KUKA KRL program: MyProgram_133().src

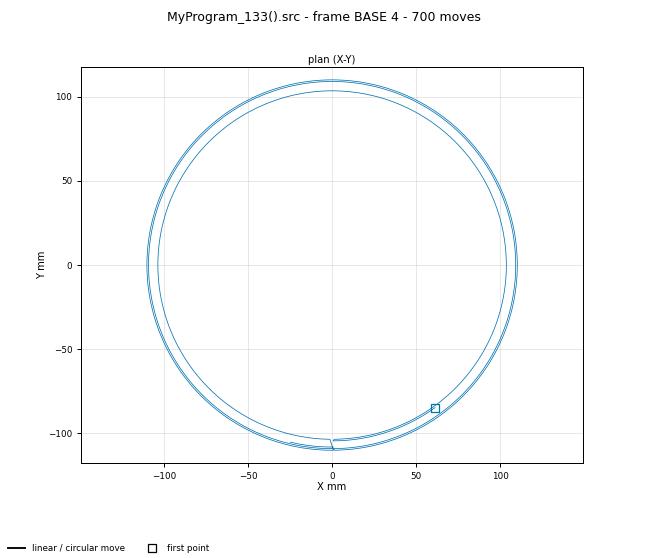
[picture p0: tool path of MyProgram_133().src in frame BASE 4, 700 of 700 moves have a stored position in this frame; points joined in program order, loops and branches not executed]
&ACCESS RVP
&REL 1
&PARAM TEMPLATE = C:\KRC\Roboter\Template\vorgabe
&PARAM EDITMASK = *
DEF MyProgram_133()
; ---- Setting reference (Base) ----
$BASE = BASE_DATA[4]

; --------------------------
; ---- Setting tool (TCP) ----
$TOOL = TOOL_DATA[3]
; --------------------------

$VEL.CP = VEL_APROX_PRINT
Startdeposition()
$VEL.CP = VEL_PRINT
LIN {X 61.2206,Y -84.8181,Z 108,A -58.6643,B 24.9452,C -1.7099,E1 25.0928,E2 504.3174} C_DIS
LIN {X 58.1513,Y -86.9519,Z 108,A -60.6312,B 24.9452,C -1.7091,E1 25.0883,E2 506.2796} C_DIS
LIN {X 55.4744,Y -88.6817,Z 108,A -62.4404,B 24.9456,C -1.7031,E1 25.084,E2 508.097} C_DIS
LIN {X 52.3012,Y -90.5896,Z 108,A -64.1698,B 24.9451,C -1.7116,E1 25.0799,E2 509.801} C_DIS
LIN {X 49.6243,Y -92.0835,Z 108,A -66.2153,B 24.9462,C -1.6936,E1 25.0748,E2 511.883} C_DIS
LIN {X 46.4014,Y -93.7484,Z 108,A -67.8646,B 24.9456,C -1.7041,E1 25.0708,E2 513.5031} C_DIS
LIN {X 42.0494,Y -95.7798,Z 108,A -71.2268,B 24.9477,C -1.6704,E1 25.0621,E2 516.9366} C_DIS
LIN {X 38.7203,Y -97.1743,Z 108,A -72.8071,B 24.9469,C -1.6835,E1 25.0581,E2 518.4823} C_DIS
LIN {X 33.6677,Y -99.0374,Z 108,A -75.7053,B 24.947,C -1.6817,E1 25.0505,E2 521.3787} C_DIS
LIN {X 30.0797,Y -100.1857,Z 108,A -77.6032,B 24.9467,C -1.6859,E1 25.0454,E2 523.2633} C_DIS
LIN {X 26.6603,Y -101.1508,Z 108,A -80.0703,B 24.9482,C -1.663,E1 25.0386,E2 525.7807} C_DIS
LIN {X 21.8993,Y -102.286,Z 108,A -82.3229,B 24.9473,C -1.6775,E1 25.0326,E2 527.9957} C_DIS
LIN {X 18.813,Y -102.8981,Z 108,A -84.0847,B 24.9475,C -1.6746,E1 25.0278,E2 529.7625} C_DIS
LIN {X 14.7921,Y -103.5522,Z 108,A -86.2883,B 24.9475,C -1.6741,E1 25.0217,E2 531.9652} C_DIS
LIN {X 12.4769,Y -103.857,Z 108,A -87.7945,B 24.9481,C -1.6643,E1 25.0174,E2 533.4935} C_DIS
LIN {X 8.4641,Y -104.2604,Z 108,A -89.7441,B 24.9475,C -1.6734,E1 25.0121,E2 535.4204} C_DIS
LIN {X 5.3432,Y -104.4676,Z 108,A -91.7149,B 24.9482,C -1.6625,E1 25.0065,E2 537.4162} C_DIS
LIN {X 0.6861,Y -104.5966,Z 108,A -93.2357,B 24.9457,C -1.7025,E1 25.0026,E2 538.842} C_DIS
Enddeposition()
LIN {X 0.6861,Y -104.5966,Z 108,A -93.2357,B 24.9457,C -1.7025,E1 25.0026,E2 538.842} C_DIS
Startdeposition()
$VEL.CP = VEL_PRINT
LIN {X 1.232,Y -103.6397,Z 108,A -93.0353,B 24.9449,C -1.715,E1 25.0032,E2 538.6119} C_DIS
LIN {X 3.4523,Y -103.5881,Z 108,A -91.8043,B 24.9449,C -1.7156,E1 25.0066,E2 537.3798} C_DIS
LIN {X 6.3528,Y -103.4523,Z 108,A -90.1987,B 24.9449,C -1.7162,E1 25.0111,E2 535.7733} C_DIS
LIN {X 8.6388,Y -103.2853,Z 108,A -88.9124,B 24.9447,C -1.7176,E1 25.0147,E2 534.4842} C_DIS
LIN {X 11.1011,Y -103.0495,Z 108,A -87.536,B 24.9447,C -1.7188,E1 25.0185,E2 533.1061} C_DIS
LIN {X 13.6424,Y -102.744,Z 108,A -86.1543,B 24.9447,C -1.7183,E1 25.0223,E2 531.7265} C_DIS
LIN {X 16.4463,Y -102.334,Z 108,A -84.5923,B 24.9447,C -1.7193,E1 25.0267,E2 530.1638} C_DIS
LIN {X 18.9681,Y -101.8968,Z 108,A -83.1777,B 24.9445,C -1.7204,E1 25.0305,E2 528.7481} C_DIS
LIN {X 21.1597,Y -101.4629,Z 108,A -81.9382,B 24.9445,C -1.7217,E1 25.0339,E2 527.5071} C_DIS
LIN {X 23.6339,Y -100.9152,Z 108,A -80.5472,B 24.9444,C -1.7226,E1 25.0377,E2 526.1158} C_DIS
LIN {X 26.3836,Y -100.2328,Z 108,A -78.9876,B 24.9444,C -1.7239,E1 25.0419,E2 524.5554} C_DIS
LIN {X 28.8655,Y -99.5466,Z 108,A -77.564,B 24.9442,C -1.7255,E1 25.0458,E2 523.1304} C_DIS
LIN {X 31.0076,Y -98.8988,Z 108,A -76.33,B 24.9442,C -1.7269,E1 25.0491,E2 521.8955} C_DIS
LIN {X 33.7061,Y -98.0134,Z 108,A -74.7661,B 24.944,C -1.7286,E1 25.0532,E2 520.3305} C_DIS
LIN {X 36.1212,Y -97.1493,Z 108,A -73.3546,B 24.9439,C -1.7302,E1 25.0569,E2 518.9182} C_DIS
LIN {X 38.4749,Y -96.2415,Z 108,A -71.9598,B 24.9438,C -1.7321,E1 25.0605,E2 517.5219} C_DIS
LIN {X 40.5286,Y -95.3932,Z 108,A -70.7044,B 24.9436,C -1.7351,E1 25.0638,E2 516.2624} C_DIS
LIN {X 42.8319,Y -94.3814,Z 108,A -69.3162,B 24.9434,C -1.7371,E1 25.0673,E2 514.8729} C_DIS
LIN {X 45.3665,Y -93.1907,Z 108,A -67.8221,B 24.9434,C -1.7374,E1 25.0711,E2 513.382} C_DIS
LIN {X 47.7293,Y -92.0036,Z 108,A -66.2293,B 24.9429,C -1.7452,E1 25.0751,E2 511.7751} C_DIS
LIN {X 50.5152,Y -90.5017,Z 108,A -64.5337,B 24.9429,C -1.7461,E1 25.0792,E2 510.0823} C_DIS
LIN {X 53.2884,Y -88.8993,Z 108,A -62.8451,B 24.9429,C -1.7459,E1 25.0833,E2 508.3992} C_DIS
LIN {X 55.1927,Y -87.7281,Z 108,A -61.613,B 24.9427,C -1.7482,E1 25.0862,E2 507.1658} C_DIS
LIN {X 57.3228,Y -86.3513,Z 108,A -60.1865,B 24.9425,C -1.7519,E1 25.0895,E2 505.7351} C_DIS
LIN {X 59.6652,Y -84.7513,Z 108,A -58.655,B 24.9424,C -1.7536,E1 25.0931,E2 504.205} C_DIS
LIN {X 61.4771,Y -83.4446,Z 108,A -57.3239,B 24.9419,C -1.7602,E1 25.0961,E2 502.863} C_DIS
LIN {X 64.262,Y -81.3187,Z 108,A -55.4103,B 24.9417,C -1.7634,E1 25.1003,E2 500.9488} C_DIS
LIN {X 67.0825,Y -79.0083,Z 108,A -53.4504,B 24.9416,C -1.7656,E1 25.1045,E2 498.9912} C_DIS
LIN {X 69.5666,Y -76.8321,Z 108,A -51.4729,B 24.9409,C -1.7762,E1 25.1087,E2 496.9967} C_DIS
LIN {X 71.9263,Y -74.6254,Z 108,A -49.8665,B 24.9411,C -1.773,E1 25.1119,E2 495.4045} C_DIS
LIN {X 74.2699,Y -72.2952,Z 108,A -47.9241,B 24.9405,C -1.7823,E1 25.1157,E2 493.4484} C_DIS
LIN {X 76.6554,Y -69.7601,Z 108,A -45.996,B 24.9401,C -1.7873,E1 25.1194,E2 491.5168} C_DIS
LIN {X 78.8973,Y -67.2128,Z 108,A -44.2153,B 24.9401,C -1.7882,E1 25.1226,E2 489.7421} C_DIS
LIN {X 81.2145,Y -64.394,Z 108,A -42.2551,B 24.9399,C -1.7912,E1 25.1261,E2 487.7839} C_DIS
LIN {X 83.0501,Y -62.009,Z 108,A -40.6111,B 24.9396,C -1.7949,E1 25.1288,E2 486.1391} C_DIS
LIN {X 85.1534,Y -59.0868,Z 108,A -38.619,B 24.9392,C -1.8005,E1 25.1321,E2 484.1435} C_DIS
LIN {X 86.8773,Y -56.525,Z 108,A -36.9669,B 24.9391,C -1.8029,E1 25.1346,E2 482.4938} C_DIS
LIN {X 88.5467,Y -53.8686,Z 108,A -35.1672,B 24.9385,C -1.8107,E1 25.1373,E2 480.6849} C_DIS
LIN {X 90.0257,Y -51.3597,Z 108,A -33.6723,B 24.9385,C -1.8105,E1 25.1393,E2 479.1981} C_DIS
LIN {X 91.265,Y -49.1238,Z 108,A -32.2106,B 24.9381,C -1.8168,E1 25.1413,E2 477.7294} C_DIS
LIN {X 92.441,Y -46.8734,Z 108,A -30.8154,B 24.9379,C -1.8206,E1 25.1431,E2 476.3325} C_DIS
LIN {X 93.5614,Y -44.595,Z 108,A -29.2927,B 24.9372,C -1.8298,E1 25.1449,E2 474.7962} C_DIS
LIN {X 95.0266,Y -41.3799,Z 108,A -27.4161,B 24.9371,C -1.8326,E1 25.1471,E2 472.9234} C_DIS
LIN {X 96.1166,Y -38.7819,Z 108,A -25.9637,B 24.9371,C -1.8329,E1 25.1486,E2 471.4781} C_DIS
LIN {X 97.1386,Y -36.1495,Z 108,A -24.4185,B 24.9367,C -1.8371,E1 25.1501,E2 469.9317} C_DIS
LIN {X 97.9881,Y -33.7787,Z 108,A -23.0399,B 24.9365,C -1.8409,E1 25.1514,E2 468.552} C_DIS
LIN {X 99.1835,Y -30.0895,Z 108,A -20.8997,B 24.936,C -1.8474,E1 25.1532,E2 466.4084} C_DIS
LIN {X 100.1166,Y -26.8152,Z 108,A -19.0121,B 24.9356,C -1.8537,E1 25.1546,E2 464.5169} C_DIS
LIN {X 100.8438,Y -23.9429,Z 108,A -17.4059,B 24.9353,C -1.8576,E1 25.1557,E2 462.9109} C_DIS
LIN {X 101.3352,Y -21.7632,Z 108,A -16.1482,B 24.935,C -1.8625,E1 25.1565,E2 461.6488} C_DIS
LIN {X 101.894,Y -18.983,Z 108,A -14.6222,B 24.9347,C -1.8658,E1 25.1573,E2 460.124} C_DIS
LIN {X 102.4789,Y -15.5091,Z 108,A -12.6574,B 24.9343,C -1.8728,E1 25.1582,E2 458.1542} C_DIS
LIN {X 102.8659,Y -12.7021,Z 108,A -11.0062,B 24.9336,C -1.8814,E1 25.1588,E2 456.4923} C_DIS
LIN {X 103.2113,Y -9.4745,Z 108,A -9.2972,B 24.9335,C -1.8837,E1 25.1592,E2 454.7882} C_DIS
LIN {X 103.4511,Y -6.3718,Z 108,A -7.6431,B 24.9333,C -1.8864,E1 25.1595,E2 453.1374} C_DIS
LIN {X 103.5758,Y -3.8438,Z 108,A -6.2514,B 24.933,C -1.8906,E1 25.1597,E2 451.744} C_DIS
LIN {X 103.6418,Y -0.8403,Z 108,A -4.5075,B 24.9324,C -1.8996,E1 25.1597,E2 449.9895} C_DIS
LIN {X 103.6218,Y 2.2287,Z 108,A -2.9186,B 24.9323,C -1.9005,E1 25.1597,E2 448.4078} C_DIS
LIN {X 103.537,Y 4.7467,Z 108,A -1.5031,B 24.9319,C -1.906,E1 25.1596,E2 446.9878} C_DIS
LIN {X 103.3869,Y 7.3217,Z 108,A -0.0895,B 24.9316,C -1.91,E1 25.1593,E2 445.5731} C_DIS
LIN {X 103.1497,Y 10.142,Z 108,A 1.4332,B 24.9314,C -1.9132,E1 25.1589,E2 444.0518} C_DIS
LIN {X 102.8676,Y 12.6886,Z 108,A 2.842,B 24.9311,C -1.9174,E1 25.1585,E2 442.6415} C_DIS
LIN {X 102.5688,Y 14.9031,Z 108,A 4.0984,B 24.9307,C -1.9223,E1 25.158,E2 441.381} C_DIS
LIN {X 102.1736,Y 17.407,Z 108,A 5.4912,B 24.9304,C -1.9263,E1 25.1573,E2 439.9869} C_DIS
LIN {X 101.7175,Y 19.8996,Z 108,A 6.8561,B 24.9302,C -1.9292,E1 25.1566,E2 438.6231} C_DIS
LIN {X 101.1284,Y 22.7109,Z 108,A 8.4288,B 24.9299,C -1.9335,E1 25.1557,E2 437.0495} C_DIS
LIN {X 100.6134,Y 24.8875,Z 108,A 9.6868,B 24.9296,C -1.9383,E1 25.1549,E2 435.7875} C_DIS
LIN {X 99.8136,Y 27.9234,Z 108,A 11.4848,B 24.929,C -1.9462,E1 25.1535,E2 433.9811} C_DIS
LIN {X 98.8964,Y 31.0154,Z 108,A 13.153,B 24.929,C -1.9468,E1 25.1522,E2 432.321} C_DIS
LIN {X 98.0105,Y 33.7149,Z 108,A 14.7133,B 24.9286,C -1.9511,E1 25.1508,E2 430.7595} C_DIS
LIN {X 97.1542,Y 36.1082,Z 108,A 16.1091,B 24.9284,C -1.9548,E1 25.1495,E2 429.3625} C_DIS
LIN {X 96.235,Y 38.4912,Z 108,A 17.5095,B 24.9281,C -1.9585,E1 25.148,E2 427.9613} C_DIS
LIN {X 95.3998,Y 40.513,Z 108,A 18.751,B 24.9277,C -1.9634,E1 25.1467,E2 426.7151} C_DIS
LIN {X 94.3673,Y 42.8631,Z 108,A 20.1553,B 24.9275,C -1.9668,E1 25.1451,E2 425.3103} C_DIS
LIN {X 93.1661,Y 45.4177,Z 108,A 21.6677,B 24.9273,C -1.9692,E1 25.1433,E2 423.8004} C_DIS
LIN {X 92.0009,Y 47.7345,Z 108,A 23.1002,B 24.927,C -1.9732,E1 25.1414,E2 422.3661} C_DIS
LIN {X 90.3319,Y 50.8193,Z 108,A 25.0281,B 24.9266,C -1.978,E1 25.1388,E2 420.4368} C_DIS
LIN {X 88.8964,Y 53.2931,Z 108,A 26.5957,B 24.9264,C -1.9817,E1 25.1366,E2 418.8686} C_DIS
LIN {X 87.729,Y 55.1913,Z 108,A 27.8136,B 24.9262,C -1.9844,E1 25.1348,E2 417.6506} C_DIS
LIN {X 86.3569,Y 57.3142,Z 108,A 29.2447,B 24.9258,C -1.9894,E1 25.1326,E2 416.2147} C_DIS
LIN {X 84.7638,Y 59.6473,Z 108,A 30.7683,B 24.9256,C -1.9918,E1 25.1302,E2 414.6931} C_DIS
LIN {X 83.428,Y 61.4998,Z 108,A 32.1191,B 24.9251,C -1.9986,E1 25.128,E2 413.3327} C_DIS
LIN {X 81.3174,Y 64.2637,Z 108,A 34.0244,B 24.9248,C -2.0026,E1 25.1247,E2 411.427} C_DIS
LIN {X 78.99,Y 67.104,Z 108,A 35.9959,B 24.9246,C -2.0049,E1 25.1212,E2 409.4589} C_DIS
LIN {X 76.9056,Y 69.4845,Z 108,A 37.7651,B 24.9243,C -2.0097,E1 25.1179,E2 407.6864} C_DIS
LIN {X 74.6426,Y 71.9085,Z 108,A 39.5541,B 24.9241,C -2.012,E1 25.1145,E2 405.8998} C_DIS
LIN {X 72.251,Y 74.3124,Z 108,A 41.5349,B 24.9235,C -2.0203,E1 25.1105,E2 403.9077} C_DIS
LIN {X 69.7041,Y 76.7068,Z 108,A 43.4992,B 24.9231,C -2.0255,E1 25.1065,E2 401.9389} C_DIS
LIN {X 67.1,Y 78.9934,Z 108,A 45.3472,B 24.923,C -2.0266,E1 25.1026,E2 400.0957} C_DIS
LIN {X 64.2763,Y 81.3075,Z 108,A 47.3173,B 24.9229,C -2.0284,E1 25.0983,E2 398.1288} C_DIS
LIN {X 61.5281,Y 83.4073,Z 108,A 49.2474,B 24.9225,C -2.0325,E1 25.094,E2 396.1959} C_DIS
LIN {X 58.8878,Y 85.2918,Z 108,A 50.9195,B 24.9227,C -2.0306,E1 25.0902,E2 394.534} C_DIS
LIN {X 56.5294,Y 86.8744,Z 108,A 52.4881,B 24.9225,C -2.0331,E1 25.0865,E2 392.9647} C_DIS
LIN {X 54.3706,Y 88.2416,Z 108,A 53.8912,B 24.9224,C -2.0349,E1 25.0832,E2 391.5618} C_DIS
LIN {X 52.4564,Y 89.3911,Z 108,A 55.2708,B 24.9218,C -2.0426,E1 25.0798,E2 390.1683} C_DIS
LIN {X 49.3867,Y 91.1224,Z 108,A 57.1622,B 24.9218,C -2.043,E1 25.0752,E2 388.2814} C_DIS
LIN {X 46.036,Y 92.8603,Z 108,A 59.213,B 24.9216,C -2.0443,E1 25.0701,E2 386.2332} C_DIS
LIN {X 43.4433,Y 94.1017,Z 108,A 60.7606,B 24.9216,C -2.0445,E1 25.0662,E2 384.689} C_DIS
LIN {X 41.1689,Y 95.1186,Z 108,A 62.1463,B 24.9215,C -2.0464,E1 25.0627,E2 383.3023} C_DIS
LIN {X 38.7671,Y 96.1227,Z 108,A 63.5401,B 24.9215,C -2.0461,E1 25.0591,E2 381.9124} C_DIS
LIN {X 36.1243,Y 97.1482,Z 108,A 65.1024,B 24.9214,C -2.0474,E1 25.055,E2 380.3504} C_DIS
LIN {X 33.9513,Y 97.9275,Z 108,A 66.3567,B 24.9214,C -2.0477,E1 25.0517,E2 379.098} C_DIS
LIN {X 31.6655,Y 98.6899,Z 108,A 67.7522,B 24.9211,C -2.0513,E1 25.048,E2 377.6965} C_DIS
LIN {X 27.9406,Y 99.8087,Z 108,A 69.8055,B 24.9213,C -2.049,E1 25.0425,E2 375.6522} C_DIS
LIN {X 25.4754,Y 100.4662,Z 108,A 71.2922,B 24.921,C -2.0529,E1 25.0385,E2 374.1586} C_DIS
LIN {X 22.7132,Y 101.1279,Z 108,A 72.8309,B 24.921,C -2.0525,E1 25.0343,E2 372.623} C_DIS
LIN {X 20.36,Y 101.6271,Z 108,A 74.1669,B 24.921,C -2.0533,E1 25.0306,E2 371.2866} C_DIS
LIN {X 18.0297,Y 102.0655,Z 108,A 75.5,B 24.9208,C -2.0547,E1 25.027,E2 369.9516} C_DIS
LIN {X 15.5027,Y 102.4799,Z 108,A 76.9132,B 24.9208,C -2.0551,E1 25.0231,E2 368.5391} C_DIS
LIN {X 12.6903,Y 102.8674,Z 108,A 78.4528,B 24.9208,C -2.0542,E1 25.0188,E2 367.0027} C_DIS
LIN {X 10.3407,Y 103.1291,Z 108,A 79.7491,B 24.9208,C -2.054,E1 25.0152,E2 365.7077} C_DIS
LIN {X 7.94,Y 103.3412,Z 108,A 81.1233,B 24.9208,C -2.0557,E1 25.0114,E2 364.3302} C_DIS
LIN {X 5.395,Y 103.5053,Z 108,A 82.5314,B 24.9208,C -2.0557,E1 25.0075,E2 362.9228} C_DIS
LIN {X 2.5412,Y 103.6161,Z 108,A 84.0795,B 24.9208,C -2.0543,E1 25.0032,E2 361.3783} C_DIS
LIN {X -0.7075,Y 103.6429,Z 108,A 85.9239,B 24.9208,C -2.0559,E1 24.998,E2 359.5303} C_DIS
LIN {X -3.491,Y 103.5869,Z 108,A 87.4167,B 24.9209,C -2.0537,E1 24.9938,E2 358.0425} C_DIS
LIN {X -6.3194,Y 103.4542,Z 108,A 88.9782,B 24.9209,C -2.0529,E1 24.9895,E2 356.4824} C_DIS
LIN {X -8.8915,Y 103.2651,Z 108,A 90.4112,B 24.9209,C -2.0525,E1 24.9855,E2 355.0496} C_DIS
LIN {X -11.1168,Y 103.0479,Z 108,A 91.6782,B 24.9209,C -2.0531,E1 24.982,E2 353.7805} C_DIS
LIN {X -13.635,Y 102.745,Z 108,A 93.0521,B 24.9211,C -2.0512,E1 24.9782,E2 352.4102} C_DIS
LIN {X -16.2113,Y 102.3703,Z 108,A 94.4883,B 24.9211,C -2.0501,E1 24.9742,E2 350.9753} C_DIS
LIN {X -18.8964,Y 101.9097,Z 108,A 95.9942,B 24.9213,C -2.0489,E1 24.9701,E2 349.4707} C_DIS
LIN {X -21.1696,Y 101.4608,Z 108,A 97.315,B 24.9213,C -2.0494,E1 24.9665,E2 348.1473} C_DIS
LIN {X -23.6474,Y 100.9121,Z 108,A 98.691,B 24.9214,C -2.0471,E1 24.9627,E2 346.7749} C_DIS
LIN {X -26.4023,Y 100.228,Z 108,A 100.2618,B 24.9215,C -2.0456,E1 24.9585,E2 345.2054} C_DIS
LIN {X -28.8474,Y 99.5517,Z 108,A 101.6638,B 24.9217,C -2.0441,E1 24.9547,E2 343.8049} C_DIS
LIN {X -32.2212,Y 98.5101,Z 108,A 103.6193,B 24.9218,C -2.042,E1 24.9495,E2 341.8508} C_DIS
LIN {X -34.6487,Y 97.6828,Z 108,A 105.0803,B 24.9218,C -2.0418,E1 24.9457,E2 340.3874} C_DIS
LIN {X -37.0274,Y 96.8061,Z 108,A 106.4832,B 24.922,C -2.04,E1 24.942,E2 338.9859} C_DIS
LIN {X -39.6631,Y 95.758,Z 108,A 108.0264,B 24.9222,C -2.0369,E1 24.938,E2 337.4466} C_DIS
LIN {X -41.9937,Y 94.759,Z 108,A 109.431,B 24.9224,C -2.0349,E1 24.9344,E2 336.0434} C_DIS
LIN {X -44.2988,Y 93.7035,Z 108,A 110.8391,B 24.9224,C -2.033,E1 24.9309,E2 334.6363} C_DIS
LIN {X -46.3069,Y 92.726,Z 108,A 112.1917,B 24.9224,C -2.0354,E1 24.9274,E2 333.2745} C_DIS
LIN {X -49.403,Y 91.1136,Z 108,A 114.0878,B 24.9227,C -2.0309,E1 24.9228,E2 331.3838} C_DIS
LIN {X -51.9345,Y 89.6954,Z 108,A 115.6552,B 24.923,C -2.0267,E1 24.919,E2 329.8217} C_DIS
LIN {X -54.3736,Y 88.2398,Z 108,A 117.2011,B 24.9233,C -2.0229,E1 24.9153,E2 328.2801} C_DIS
LIN {X -56.2655,Y 87.0439,Z 108,A 118.4438,B 24.9234,C -2.0208,E1 24.9124,E2 327.0385} C_DIS
LIN {X -58.1444,Y 85.7996,Z 108,A 119.7907,B 24.9234,C -2.022,E1 24.9093,E2 325.6841} C_DIS
LIN {X -60.7085,Y 84.0072,Z 108,A 121.4301,B 24.9239,C -2.0152,E1 24.9055,E2 324.0553} C_DIS
LIN {X -62.8831,Y 82.3911,Z 108,A 123.0928,B 24.9236,C -2.0181,E1 24.9018,E2 322.3798} C_DIS
LIN {X -65.6338,Y 80.2171,Z 108,A 125.0735,B 24.9238,C -2.0154,E1 24.8975,E2 320.3981} C_DIS
LIN {X -68.172,Y 78.0699,Z 108,A 126.8213,B 24.9244,C -2.008,E1 24.8938,E2 318.6611} C_DIS
LIN {X -70.6386,Y 75.8471,Z 108,A 128.7417,B 24.9244,C -2.0068,E1 24.8899,E2 316.7358} C_DIS
LIN {X -72.9443,Y 73.6308,Z 108,A 130.4853,B 24.9249,C -2.0017,E1 24.8864,E2 314.9971} C_DIS
LIN {X -75.4965,Y 71.0114,Z 108,A 132.4762,B 24.9253,C -1.9956,E1 24.8826,E2 313.0121} C_DIS
LIN {X -77.9537,Y 68.3051,Z 108,A 134.5012,B 24.9257,C -1.9906,E1 24.8788,E2 310.99} C_DIS
LIN {X -80.2153,Y 65.636,Z 108,A 136.5204,B 24.9259,C -1.9886,E1 24.8752,E2 308.9662} C_DIS
LIN {X -82.3897,Y 62.8848,Z 108,A 138.3219,B 24.9266,C -1.9785,E1 24.8721,E2 307.1802} C_DIS
LIN {X -84.318,Y 60.273,Z 108,A 140.1752,B 24.9268,C -1.9757,E1 24.8691,E2 305.3245} C_DIS
LIN {X -86.0119,Y 57.8309,Z 108,A 141.8008,B 24.9272,C -1.9705,E1 24.8665,E2 303.7033} C_DIS
LIN {X -87.5654,Y 55.4531,Z 108,A 143.3517,B 24.9276,C -1.9654,E1 24.8642,E2 302.1568} C_DIS
LIN {X -88.7411,Y 53.5488,Z 108,A 144.5964,B 24.9278,C -1.9621,E1 24.8624,E2 300.9135} C_DIS
LIN {X -90.1876,Y 51.0778,Z 108,A 146.1839,B 24.9281,C -1.9577,E1 24.8602,E2 299.3283} C_DIS
LIN {X -91.2533,Y 49.1455,Z 108,A 147.4468,B 24.9283,C -1.9557,E1 24.8585,E2 298.0636} C_DIS
LIN {X -92.4104,Y 46.9332,Z 108,A 148.8392,B 24.9286,C -1.952,E1 24.8567,E2 296.6724} C_DIS
LIN {X -94.0137,Y 43.6324,Z 108,A 150.8777,B 24.929,C -1.9463,E1 24.8543,E2 294.6366} C_DIS
LIN {X -95.1432,Y 41.1124,Z 108,A 152.4143,B 24.9293,C -1.942,E1 24.8525,E2 293.1017} C_DIS
LIN {X -96.1213,Y 38.7704,Z 108,A 153.7973,B 24.9297,C -1.937,E1 24.8511,E2 291.7229} C_DIS
LIN {X -97.1484,Y 36.1237,Z 108,A 155.3757,B 24.93,C -1.9324,E1 24.8495,E2 290.1465} C_DIS
LIN {X -98.0035,Y 33.7347,Z 108,A 156.9137,B 24.93,C -1.9328,E1 24.8481,E2 288.5988} C_DIS
LIN {X -99.0404,Y 30.5511,Z 108,A 158.7275,B 24.9305,C -1.9257,E1 24.8466,E2 286.7915} C_DIS
LIN {X -99.8126,Y 27.9268,Z 108,A 160.2069,B 24.9309,C -1.9198,E1 24.8454,E2 285.3177} C_DIS
LIN {X -100.4668,Y 25.4733,Z 108,A 161.62,B 24.9312,C -1.9157,E1 24.8444,E2 283.9063} C_DIS
LIN {X -101.1288,Y 22.7093,Z 108,A 163.1719,B 24.9316,C -1.91,E1 24.8435,E2 282.3588} C_DIS
LIN {X -101.6489,Y 20.2534,Z 108,A 164.57,B 24.9319,C -1.9059,E1 24.8427,E2 280.9622} C_DIS
LIN {X -102.2143,Y 17.1636,Z 108,A 166.4073,B 24.932,C -1.9039,E1 24.8418,E2 279.1188} C_DIS
LIN {X -102.7052,Y 13.9424,Z 108,A 168.1309,B 24.9327,C -1.8953,E1 24.8411,E2 277.4054} C_DIS
LIN {X -103.0159,Y 11.4226,Z 108,A 169.7522,B 24.9324,C -1.8985,E1 24.8406,E2 275.7668} C_DIS
LIN {X -103.3419,Y 7.9308,Z 108,A 171.5279,B 24.9333,C -1.8865,E1 24.8402,E2 274.0091} C_DIS
LIN {X -103.5549,Y 4.3293,Z 108,A 173.5851,B 24.9336,C -1.8822,E1 24.8399,E2 271.9497} C_DIS
LIN {X -103.642,Y 0.7964,Z 108,A 175.5561,B 24.934,C -1.8765,E1 24.8398,E2 269.9804} C_DIS
LIN {X -103.6217,Y -2.2357,Z 108,A 177.162,B 24.9345,C -1.8686,E1 24.8398,E2 268.3836} C_DIS
LIN {X -103.5057,Y -5.3879,Z 108,A 179.0297,B 24.9346,C -1.8674,E1 24.8401,E2 266.5076} C_DIS
LIN {X -103.2647,Y -8.896,Z 108,A -179.1251,B 24.9353,C -1.8577,E1 24.8405,E2 264.6746} C_DIS
LIN {X -103.0472,Y -11.1234,Z 108,A -177.8482,B 24.9355,C -1.8551,E1 24.8408,E2 263.3959} C_DIS
LIN {X -102.7438,Y -13.6445,Z 108,A -176.3065,B 24.9355,C -1.8556,E1 24.8414,E2 261.844} C_DIS
LIN {X -102.2142,Y -17.164,Z 108,A -174.3931,B 24.936,C -1.8475,E1 24.8422,E2 259.9386} C_DIS
LIN {X -101.7122,Y -19.9271,Z 108,A -172.9207,B 24.9366,C -1.8397,E1 24.843,E2 258.476} C_DIS
LIN {X -101.1293,Y -22.707,Z 108,A -171.3398,B 24.9369,C -1.8352,E1 24.8439,E2 256.8965} C_DIS
LIN {X -100.6141,Y -24.8848,Z 108,A -170.1401,B 24.9372,C -1.8301,E1 24.8447,E2 255.702} C_DIS
LIN {X -99.9702,Y -27.3571,Z 108,A -168.6422,B 24.9373,C -1.8288,E1 24.8458,E2 254.1985} C_DIS
LIN {X -99.2646,Y -29.8162,Z 108,A -167.2498,B 24.9377,C -1.8237,E1 24.8469,E2 252.8101} C_DIS
LIN {X -98.5091,Y -32.2245,Z 108,A -165.8153,B 24.9378,C -1.8209,E1 24.8481,E2 251.374} C_DIS
LIN {X -97.6951,Y -34.6138,Z 108,A -164.4337,B 24.9382,C -1.8163,E1 24.8494,E2 249.9957} C_DIS
LIN {X -96.8086,Y -37.0211,Z 108,A -162.9832,B 24.9384,C -1.8133,E1 24.8508,E2 248.5442} C_DIS
LIN {X -95.7599,Y -39.6584,Z 108,A -161.3123,B 24.9384,C -1.8123,E1 24.8526,E2 246.8663} C_DIS
LIN {X -94.475,Y -42.6241,Z 108,A -159.5992,B 24.939,C -1.8046,E1 24.8545,E2 245.1622} C_DIS
LIN {X -93.1441,Y -45.4634,Z 108,A -157.8921,B 24.9394,C -1.7987,E1 24.8565,E2 243.4598} C_DIS
LIN {X -92.0025,Y -47.7314,Z 108,A -156.4787,B 24.9396,C -1.7952,E1 24.8583,E2 242.0472} C_DIS
LIN {X -90.5367,Y -50.4525,Z 108,A -154.7036,B 24.9397,C -1.793,E1 24.8607,E2 240.2682} C_DIS
LIN {X -88.9024,Y -53.2833,Z 108,A -152.9424,B 24.9402,C -1.7864,E1 24.8632,E2 238.5133} C_DIS
LIN {X -87.7312,Y -55.1877,Z 108,A -151.7,B 24.9404,C -1.7835,E1 24.865,E2 237.2717} C_DIS
LIN {X -85.9512,Y -57.9205,Z 108,A -149.8005,B 24.9404,C -1.7823,E1 24.868,E2 235.3654} C_DIS
LIN {X -84.0017,Y -60.7163,Z 108,A -147.9917,B 24.941,C -1.7748,E1 24.8709,E2 233.5656} C_DIS
LIN {X -82.3878,Y -62.8874,Z 108,A -146.3337,B 24.9408,C -1.7771,E1 24.8737,E2 231.8943} C_DIS
LIN {X -80.215,Y -65.6364,Z 108,A -144.3522,B 24.941,C -1.7741,E1 24.8772,E2 229.9106} C_DIS
LIN {X -78.069,Y -68.1731,Z 108,A -142.6057,B 24.9415,C -1.7666,E1 24.8803,E2 228.174} C_DIS
LIN {X -75.8267,Y -70.6603,Z 108,A -140.7359,B 24.9417,C -1.7631,E1 24.8839,E2 226.3042} C_DIS
LIN {X -73.6376,Y -72.9374,Z 108,A -138.9551,B 24.9419,C -1.7607,E1 24.8874,E2 224.5217} C_DIS
LIN {X -71.0306,Y -75.4784,Z 108,A -136.9595,B 24.9422,C -1.7559,E1 24.8914,E2 222.5292} C_DIS
LIN {X -68.2943,Y -77.9632,Z 108,A -134.9648,B 24.9426,C -1.75,E1 24.8955,E2 220.5405} C_DIS
LIN {X -65.8787,Y -80.016,Z 108,A -133.0599,B 24.9425,C -1.7523,E1 24.8996,E2 218.6229} C_DIS
LIN {X -63.267,Y -82.0952,Z 108,A -131.3258,B 24.9429,C -1.7449,E1 24.9034,E2 216.9001} C_DIS
LIN {X -60.7201,Y -83.9989,Z 108,A -129.6302,B 24.9433,C -1.7395,E1 24.9072,E2 215.2113} C_DIS
LIN {X -58.8767,Y -85.2994,Z 108,A -128.3783,B 24.9434,C -1.7376,E1 24.9101,E2 213.9596} C_DIS
LIN {X -56.5214,Y -86.8797,Z 108,A -126.8042,B 24.9436,C -1.7353,E1 24.9137,E2 212.3858} C_DIS
LIN {X -53.5528,Y -88.7386,Z 108,A -124.8622,B 24.9437,C -1.7326,E1 24.9184,E2 210.4441} C_DIS
LIN {X -51.0885,Y -90.1816,Z 108,A -123.2781,B 24.9439,C -1.7306,E1 24.9222,E2 208.8602} C_DIS
LIN {X -49.1281,Y -91.2627,Z 108,A -122.0074,B 24.9439,C -1.7302,E1 24.9253,E2 207.5868} C_DIS
LIN {X -46.8754,Y -92.4399,Z 108,A -120.5982,B 24.944,C -1.7286,E1 24.9288,E2 206.1776} C_DIS
LIN {X -44.5972,Y -93.5604,Z 108,A -119.2186,B 24.9442,C -1.726,E1 24.9323,E2 204.8007} C_DIS
LIN {X -42.0022,Y -94.7553,Z 108,A -117.6375,B 24.9442,C -1.7243,E1 24.9363,E2 203.2198} C_DIS
LIN {X -39.6722,Y -95.7541,Z 108,A -116.2342,B 24.9444,C -1.7229,E1 24.9399,E2 201.8165} C_DIS
LIN {X -37.5987,Y -96.5856,Z 108,A -115.021,B 24.9445,C -1.7209,E1 24.9431,E2 200.6055} C_DIS
LIN {X -35.3019,Y -97.4483,Z 108,A -113.6114,B 24.9445,C -1.7217,E1 24.9468,E2 199.1911} C_DIS
LIN {X -32.8945,Y -98.2871,Z 108,A -112.1761,B 24.9445,C -1.7215,E1 24.9506,E2 197.7534} C_DIS
LIN {X -30.0962,Y -99.1814,Z 108,A -110.5959,B 24.9446,C -1.7186,E1 24.9548,E2 196.1774} C_DIS
LIN {X -27.9323,Y -99.811,Z 108,A -109.3215,B 24.9446,C -1.7189,E1 24.9582,E2 194.9002} C_DIS
LIN {X -25.4791,Y -100.4653,Z 108,A -107.9155,B 24.9446,C -1.7182,E1 24.962,E2 193.4939} C_DIS
LIN {X -22.7173,Y -101.127,Z 108,A -106.3746,B 24.9448,C -1.7162,E1 24.9662,E2 191.9556} C_DIS
LIN {X -20.2338,Y -101.653,Z 108,A -104.9684,B 24.9448,C -1.7157,E1 24.97,E2 190.5489} C_DIS
LIN {X -18.0137,Y -102.0684,Z 108,A -103.6904,B 24.9448,C -1.7165,E1 24.9736,E2 189.2678} C_DIS
LIN {X -15.51,Y -102.4787,Z 108,A -102.286,B 24.9448,C -1.7162,E1 24.9774,E2 187.8629} C_DIS
LIN {X -12.6987,Y -102.8663,Z 108,A -100.7478,B 24.9449,C -1.7147,E1 24.9817,E2 186.3272} C_DIS
LIN {X -9.2,Y -103.2367,Z 108,A -98.8016,B 24.9449,C -1.7145,E1 24.9871,E2 184.3801} C_DIS
LIN {X -6.374,Y -103.4509,Z 108,A -97.2366,B 24.9449,C -1.7145,E1 24.9914,E2 182.8147} C_DIS
LIN {X -3.8214,Y -103.5767,Z 108,A -95.8215,B 24.9449,C -1.7147,E1 24.9954,E2 181.3989} C_DIS
LIN {X -1.2939,Y -103.639,Z 108,A -94.4279,B 24.9449,C -1.7147,E1 24.9993,E2 180.005} C_DIS
LIN {X -1.2939,Y -103.639,Z 108,A -94.4279,B 24.9449,C -1.7147,E1 24.9993,E2 180.005} C_DIS
Enddeposition()
LIN {X 0.7653,Y -110.1586,Z 109,A -93.3798,B 24.9517,C -1.606,E1 25.0015,E2 179.2148} C_DIS
Startdeposition()
$VEL.CP = VEL_PRINT
LIN {X -1.1992,Y -110.1569,Z 109,A -94.7506,B 24.9526,C -1.5911,E1 24.9976,E2 180.6209} C_DIS
LIN {X -3.9022,Y -110.0943,Z 109,A -96.1565,B 24.9526,C -1.5909,E1 24.9936,E2 182.0273} C_DIS
LIN {X -6.556,Y -109.9679,Z 109,A -97.5338,B 24.9526,C -1.591,E1 24.9898,E2 183.4048} C_DIS
LIN {X -9.4518,Y -109.758,Z 109,A -99.0407,B 24.9526,C -1.5912,E1 24.9856,E2 184.912} C_DIS
LIN {X -11.9907,Y -109.5089,Z 109,A -100.3754,B 24.9526,C -1.591,E1 24.9819,E2 186.2478} C_DIS
LIN {X -14.826,Y -109.162,Z 109,A -101.854,B 24.9526,C -1.5916,E1 24.9778,E2 187.7262} C_DIS
LIN {X -17.2554,Y -108.8032,Z 109,A -103.1504,B 24.9526,C -1.5911,E1 24.9742,E2 189.0248} C_DIS
LIN {X -20.0142,Y -108.3301,Z 109,A -104.5964,B 24.9526,C -1.592,E1 24.9702,E2 190.4701} C_DIS
LIN {X -22.6667,Y -107.8063,Z 109,A -106.0039,B 24.9525,C -1.5926,E1 24.9664,E2 191.878} C_DIS
LIN {X -25.4543,Y -107.1832,Z 109,A -107.4835,B 24.9525,C -1.5935,E1 24.9624,E2 193.3572} C_DIS
LIN {X -28.0771,Y -106.5262,Z 109,A -108.8918,B 24.9524,C -1.5943,E1 24.9586,E2 194.7658} C_DIS
LIN {X -30.6829,Y -105.8051,Z 109,A -110.3,B 24.9524,C -1.5951,E1 24.9548,E2 196.1742} C_DIS
LIN {X -33.1244,Y -105.0655,Z 109,A -111.6363,B 24.9523,C -1.5957,E1 24.9512,E2 197.5114} C_DIS
LIN {X -35.6929,Y -104.2209,Z 109,A -113.0089,B 24.9521,C -1.5982,E1 24.9476,E2 198.8806} C_DIS
LIN {X -38.2398,Y -103.3136,Z 109,A -114.4542,B 24.9521,C -1.5979,E1 24.9438,E2 200.3297} C_DIS
LIN {X -40.7637,Y -102.344,Z 109,A -115.8633,B 24.9521,C -1.5991,E1 24.9401,E2 201.7389} C_DIS
LIN {X -43.2631,Y -101.3128,Z 109,A -117.2654,B 24.952,C -1.6008,E1 24.9365,E2 203.1402} C_DIS
LIN {X -45.7364,Y -100.2205,Z 109,A -118.6823,B 24.952,C -1.6019,E1 24.9329,E2 204.5579} C_DIS
LIN {X -48.3198,Y -99.0018,Z 109,A -120.1644,B 24.9518,C -1.6038,E1 24.9292,E2 206.0392} C_DIS
LIN {X -50.5989,Y -97.8556,Z 109,A -121.4949,B 24.9518,C -1.6054,E1 24.9259,E2 207.3697} C_DIS
LIN {X -52.638,Y -96.7727,Z 109,A -122.7743,B 24.9518,C -1.6038,E1 24.9227,E2 208.6563} C_DIS
LIN {X -55.4719,Y -95.1789,Z 109,A -124.3953,B 24.9515,C -1.609,E1 24.9188,E2 210.2698} C_DIS
LIN {X -57.6605,Y -93.8682,Z 109,A -125.7339,B 24.9515,C -1.6105,E1 24.9156,E2 211.609} C_DIS
LIN {X -59.9468,Y -92.4249,Z 109,A -127.1375,B 24.9513,C -1.6128,E1 24.9123,E2 213.0117} C_DIS
LIN {X -62.197,Y -90.9259,Z 109,A -128.5486,B 24.9511,C -1.6149,E1 24.909,E2 214.4225} C_DIS
LIN {X -64.534,Y -89.2834,Z 109,A -130.0396,B 24.951,C -1.6172,E1 24.9056,E2 215.9132} C_DIS
LIN {X -66.7057,Y -87.6728,Z 109,A -131.4514,B 24.9509,C -1.6194,E1 24.9025,E2 217.3247} C_DIS
LIN {X -68.7174,Y -86.104,Z 109,A -132.7835,B 24.9507,C -1.6216,E1 24.8995,E2 218.6564} C_DIS
LIN {X -70.8098,Y -84.3917,Z 109,A -134.203,B 24.9506,C -1.6238,E1 24.8965,E2 220.0763} C_DIS
LIN {X -72.9745,Y -82.528,Z 109,A -135.6873,B 24.9504,C -1.6267,E1 24.8934,E2 221.5594} C_DIS
LIN {X -74.8654,Y -80.8155,Z 109,A -137.0276,B 24.9503,C -1.6289,E1 24.8906,E2 222.9} C_DIS
LIN {X -76.9361,Y -78.8479,Z 109,A -138.5128,B 24.9501,C -1.632,E1 24.8876,E2 224.3839} C_DIS
LIN {X -78.7406,Y -77.0447,Z 109,A -139.8158,B 24.9499,C -1.6358,E1 24.8851,E2 225.6834} C_DIS
LIN {X -80.6077,Y -75.0891,Z 109,A -141.2608,B 24.9498,C -1.6374,E1 24.8823,E2 227.131} C_DIS
LIN {X -82.528,Y -72.9745,Z 109,A -142.7513,B 24.9496,C -1.6405,E1 24.8795,E2 228.6206} C_DIS
LIN {X -84.195,Y -71.0435,Z 109,A -144.0759,B 24.9494,C -1.6437,E1 24.8771,E2 229.9437} C_DIS
LIN {X -86.0093,Y -68.8372,Z 109,A -145.5783,B 24.9492,C -1.6465,E1 24.8745,E2 231.4463} C_DIS
LIN {X -87.5796,Y -66.8266,Z 109,A -146.912,B 24.949,C -1.6495,E1 24.8722,E2 232.7792} C_DIS
LIN {X -89.1932,Y -64.6572,Z 109,A -148.3257,B 24.9488,C -1.6527,E1 24.8699,E2 234.1922} C_DIS
LIN {X -90.8402,Y -62.3234,Z 109,A -149.8197,B 24.9486,C -1.6561,E1 24.8675,E2 235.6854} C_DIS
LIN {X -92.3424,Y -60.0753,Z 109,A -151.2338,B 24.9484,C -1.6594,E1 24.8653,E2 237.0987} C_DIS
LIN {X -93.708,Y -57.9205,Z 109,A -152.5756,B 24.9482,C -1.6624,E1 24.8633,E2 238.4404} C_DIS
LIN {X -95.1012,Y -55.6034,Z 109,A -153.9826,B 24.948,C -1.6661,E1 24.8613,E2 239.8457} C_DIS
LIN {X -96.4371,Y -53.2527,Z 109,A -155.4047,B 24.9478,C -1.6693,E1 24.8594,E2 241.2676} C_DIS
LIN {X -97.7861,Y -50.7349,Z 109,A -156.8915,B 24.9475,C -1.6733,E1 24.8574,E2 242.7528} C_DIS
LIN {X -98.8111,Y -48.7044,Z 109,A -158.1168,B 24.9475,C -1.6751,E1 24.8559,E2 243.9805} C_DIS
LIN {X -100.0934,Y -46.0141,Z 109,A -159.649,B 24.9471,C -1.6801,E1 24.8541,E2 245.509} C_DIS
LIN {X -101.2535,Y -43.4038,Z 109,A -161.1367,B 24.9468,C -1.6843,E1 24.8524,E2 246.9949} C_DIS
LIN {X -102.2306,Y -41.0473,Z 109,A -162.4795,B 24.9466,C -1.6876,E1 24.851,E2 248.3374} C_DIS
LIN {X -103.2072,Y -38.5261,Z 109,A -163.8917,B 24.9464,C -1.6915,E1 24.8496,E2 249.7482} C_DIS
LIN {X -104.1721,Y -35.8376,Z 109,A -165.3821,B 24.9461,C -1.6957,E1 24.8482,E2 251.237} C_DIS
LIN {X -104.8982,Y -33.6475,Z 109,A -166.6331,B 24.9461,C -1.6974,E1 24.8472,E2 252.4911} C_DIS
LIN {X -105.7617,Y -30.8293,Z 109,A -168.1335,B 24.9456,C -1.7033,E1 24.846,E2 253.9861} C_DIS
LIN {X -106.4864,Y -28.2245,Z 109,A -169.549,B 24.9454,C -1.7073,E1 24.8449,E2 255.4004} C_DIS
LIN {X -107.1832,Y -25.4543,Z 109,A -171.0444,B 24.9451,C -1.7115,E1 24.8439,E2 256.8945} C_DIS
LIN {X -107.743,Y -22.9655,Z 109,A -172.3879,B 24.9449,C -1.715,E1 24.8431,E2 258.2375} C_DIS
LIN {X -108.2742,Y -20.3144,Z 109,A -173.8025,B 24.9446,C -1.7191,E1 24.8424,E2 259.6507} C_DIS
LIN {X -108.7401,Y -17.6511,Z 109,A -175.2197,B 24.9444,C -1.7231,E1 24.8417,E2 261.0667} C_DIS
LIN {X -109.162,Y -14.826,Z 109,A -176.7082,B 24.9441,C -1.7277,E1 24.8411,E2 262.5532} C_DIS
LIN {X -109.4752,Y -12.2942,Z 109,A -178.0519,B 24.9438,C -1.7313,E1 24.8407,E2 263.8963} C_DIS
LIN {X -109.744,Y -9.6039,Z 109,A -179.4603,B 24.9435,C -1.7357,E1 24.8403,E2 265.3027} C_DIS
LIN {X -109.9569,Y -6.7554,Z 109,A 179.0437,B 24.9433,C -1.7401,E1 24.84,E2 266.7972} C_DIS
LIN {X -110.083,Y -4.2074,Z 109,A 177.6999,B 24.943,C -1.7438,E1 24.8399,E2 268.1404} C_DIS
LIN {X -110.16,Y -0.7615,Z 109,A 175.8672,B 24.9427,C -1.7481,E1 24.8398,E2 269.9739} C_DIS
LIN {X -110.1311,Y 2.7036,Z 109,A 174.0876,B 24.9423,C -1.7547,E1 24.8398,E2 271.7483} C_DIS
LIN {X -110.0315,Y 5.4055,Z 109,A 172.671,B 24.942,C -1.7589,E1 24.84,E2 273.1635} C_DIS
LIN {X -109.876,Y 7.9518,Z 109,A 171.3351,B 24.9418,C -1.7629,E1 24.8403,E2 274.498} C_DIS
LIN {X -109.6338,Y 10.798,Z 109,A 169.839,B 24.9415,C -1.7673,E1 24.8407,E2 275.9925} C_DIS
LIN {X -109.3357,Y 13.4853,Z 109,A 168.4226,B 24.9412,C -1.7714,E1 24.8411,E2 277.4075} C_DIS
LIN {X -108.9934,Y 16.0133,Z 109,A 167.0789,B 24.9409,C -1.7751,E1 24.8416,E2 278.7505} C_DIS
LIN {X -108.5424,Y 18.8339,Z 109,A 165.5904,B 24.9406,C -1.7798,E1 24.8423,E2 280.2367} C_DIS
LIN {X -108.0475,Y 21.492,Z 109,A 164.1742,B 24.9404,C -1.7839,E1 24.8431,E2 281.6513} C_DIS
LIN {X -107.4875,Y 24.1371,Z 109,A 162.758,B 24.9401,C -1.788,E1 24.8439,E2 283.0661} C_DIS
LIN {X -106.8989,Y 26.6194,Z 109,A 161.4145,B 24.9398,C -1.7917,E1 24.8448,E2 284.4087} C_DIS
LIN {X -106.1737,Y 29.3822,Z 109,A 159.9262,B 24.9395,C -1.7963,E1 24.8459,E2 285.8948} C_DIS
LIN {X -105.464,Y 31.8326,Z 109,A 158.5828,B 24.9393,C -1.7999,E1 24.8469,E2 287.2373} C_DIS
LIN {X -104.6511,Y 34.4112,Z 109,A 157.1668,B 24.939,C -1.8039,E1 24.8481,E2 288.6518} C_DIS
LIN {X -103.775,Y 36.9691,Z 109,A 155.751,B 24.9387,C -1.8079,E1 24.8494,E2 290.0661} C_DIS
LIN {X -102.8365,Y 39.5048,Z 109,A 154.3426,B 24.9384,C -1.8122,E1 24.8508,E2 291.4722} C_DIS
LIN {X -101.8361,Y 42.0166,Z 109,A 152.955,B 24.9381,C -1.8172,E1 24.8523,E2 292.8556} C_DIS
LIN {X -100.7132,Y 44.6431,Z 109,A 151.4316,B 24.9379,C -1.8203,E1 24.854,E2 294.3799} C_DIS
LIN {X -99.5873,Y 47.1013,Z 109,A 150.0162,B 24.9376,C -1.8242,E1 24.8556,E2 295.7938} C_DIS
LIN {X -98.4692,Y 49.3943,Z 109,A 148.6806,B 24.9374,C -1.8279,E1 24.8573,E2 297.1279} C_DIS
LIN {X -97.1562,Y 51.9311,Z 109,A 147.1855,B 24.9371,C -1.8319,E1 24.8592,E2 298.6213} C_DIS
LIN {X -95.9269,Y 54.1664,Z 109,A 145.8502,B 24.9369,C -1.8355,E1 24.861,E2 299.9552} C_DIS
LIN {X -94.5687,Y 56.5043,Z 109,A 144.435,B 24.9366,C -1.8392,E1 24.863,E2 301.3688} C_DIS
LIN {X -93.0726,Y 58.9376,Z 109,A 142.9402,B 24.9363,C -1.8431,E1 24.8652,E2 302.862} C_DIS
LIN {X -91.7362,Y 60.9947,Z 109,A 141.6377,B 24.9361,C -1.8457,E1 24.8672,E2 304.1649} C_DIS
LIN {X -90.1677,Y 63.2909,Z 109,A 140.1918,B 24.9359,C -1.8497,E1 24.8695,E2 305.6083} C_DIS
LIN {X -88.4847,Y 65.6248,Z 109,A 138.6961,B 24.9356,C -1.8538,E1 24.872,E2 307.1014} C_DIS
LIN {X -86.8476,Y 67.7765,Z 109,A 137.2815,B 24.9353,C -1.8572,E1 24.8744,E2 308.5146} C_DIS
LIN {X -85.2543,Y 69.7688,Z 109,A 135.9469,B 24.9351,C -1.8605,E1 24.8767,E2 309.8477} C_DIS
LIN {X -83.4173,Y 71.9563,Z 109,A 134.4532,B 24.9349,C -1.864,E1 24.8794,E2 311.3399} C_DIS
LIN {X -80.8155,Y 74.8654,Z 109,A 132.4119,B 24.9345,C -1.8687,E1 24.8833,E2 313.379} C_DIS
LIN {X -78.9539,Y 76.8261,Z 109,A 130.9981,B 24.9343,C -1.8719,E1 24.886,E2 314.7913} C_DIS
LIN {X -77.0447,Y 78.7406,Z 109,A 129.5844,B 24.9341,C -1.875,E1 24.8888,E2 316.2035} C_DIS
LIN {X -75.0891,Y 80.6077,Z 109,A 128.1711,B 24.9339,C -1.8781,E1 24.8917,E2 317.6154} C_DIS
LIN {X -73.0883,Y 82.4262,Z 109,A 126.7577,B 24.9337,C -1.881,E1 24.8946,E2 319.0273} C_DIS
LIN {X -71.0435,Y 84.195,Z 109,A 125.3445,B 24.9335,C -1.8839,E1 24.8976,E2 320.4392} C_DIS
LIN {X -68.8372,Y 86.0093,Z 109,A 123.8519,B 24.9333,C -1.8869,E1 24.9008,E2 321.9302} C_DIS
LIN {X -66.8266,Y 87.5796,Z 109,A 122.5188,B 24.9331,C -1.8895,E1 24.9038,E2 323.262} C_DIS
LIN {X -64.6572,Y 89.1932,Z 109,A 121.1063,B 24.9329,C -1.8922,E1 24.9069,E2 324.6731} C_DIS
LIN {X -62.3234,Y 90.8402,Z 109,A 119.614,B 24.9327,C -1.8949,E1 24.9104,E2 326.164} C_DIS
LIN {X -60.0753,Y 92.3424,Z 109,A 118.2019,B 24.9325,C -1.8974,E1 24.9137,E2 327.5749} C_DIS
LIN {X -57.791,Y 93.7889,Z 109,A 116.7902,B 24.9323,C -1.8999,E1 24.917,E2 328.9852} C_DIS
LIN {X -55.8112,Y 94.9783,Z 109,A 115.5554,B 24.9323,C -1.9008,E1 24.92,E2 330.2216} C_DIS
LIN {X -53.2527,Y 96.4371,Z 109,A 114.0387,B 24.932,C -1.904,E1 24.9236,E2 331.7349} C_DIS
LIN {X -49.7963,Y 98.2659,Z 109,A 111.9793,B 24.9319,C -1.9064,E1 24.9287,E2 333.7943} C_DIS
LIN {X -47.1013,Y 99.5873,Z 109,A 110.4385,B 24.9316,C -1.9097,E1 24.9326,E2 335.3314} C_DIS
LIN {X -44.6431,Y 100.7132,Z 109,A 109.0277,B 24.9315,C -1.9116,E1 24.9362,E2 336.741} C_DIS
LIN {X -42.158,Y 101.7785,Z 109,A 107.6172,B 24.9314,C -1.9135,E1 24.9398,E2 338.1503} C_DIS
LIN {X -39.6476,Y 102.7824,Z 109,A 106.2068,B 24.9312,C -1.9152,E1 24.9435,E2 339.5596} C_DIS
LIN {X -37.1132,Y 103.7245,Z 109,A 104.7961,B 24.9312,C -1.9169,E1 24.9472,E2 340.9692} C_DIS
LIN {X -34.5565,Y 104.604,Z 109,A 103.3863,B 24.931,C -1.9184,E1 24.9509,E2 342.378} C_DIS
LIN {X -31.979,Y 105.4206,Z 109,A 101.9766,B 24.9309,C -1.9199,E1 24.9547,E2 343.7866} C_DIS
LIN {X -29.5291,Y 106.132,Z 109,A 100.6467,B 24.9309,C -1.9212,E1 24.9582,E2 345.1155} C_DIS
LIN {X -26.9156,Y 106.8247,Z 109,A 99.2387,B 24.9307,C -1.9226,E1 24.962,E2 346.5224} C_DIS
LIN {X -24.2859,Y 107.4531,Z 109,A 97.8282,B 24.9307,C -1.9237,E1 24.9659,E2 347.932} C_DIS
LIN {X -21.492,Y 108.0475,Z 109,A 96.34,B 24.9305,C -1.9248,E1 24.9699,E2 349.4194} C_DIS
LIN {X -18.8339,Y 108.5424,Z 109,A 94.9315,B 24.9305,C -1.9258,E1 24.9738,E2 350.8269} C_DIS
LIN {X -16.1645,Y 108.9719,Z 109,A 93.5229,B 24.9305,C -1.9267,E1 24.9777,E2 352.2347} C_DIS
LIN {X -13.7663,Y 109.2993,Z 109,A 92.2507,B 24.9304,C -1.9269,E1 24.9812,E2 353.5072} C_DIS
LIN {X -10.9499,Y 109.6179,Z 109,A 90.7867,B 24.9304,C -1.9281,E1 24.9853,E2 354.9693} C_DIS
LIN {X -8.2564,Y 109.8536,Z 109,A 89.3716,B 24.9303,C -1.9284,E1 24.9892,E2 356.3843} C_DIS
LIN {X -5.558,Y 110.0231,Z 109,A 87.9716,B 24.9303,C -1.9292,E1 24.9931,E2 357.7829} C_DIS
LIN {X -2.7036,Y 110.1311,Z 109,A 86.4852,B 24.9302,C -1.9296,E1 24.9973,E2 359.2686} C_DIS
LIN {X 0,Y 110.1642,Z 109,A 85.0782,B 24.9302,C -1.9299,E1 25.0012,E2 360.675} C_DIS
LIN {X 2.7036,Y 110.1311,Z 109,A 83.6717,B 24.9302,C -1.9301,E1 25.0051,E2 362.0807} C_DIS
LIN {X 5.4055,Y 110.0315,Z 109,A 82.2649,B 24.9302,C -1.9301,E1 25.009,E2 363.4871} C_DIS
LIN {X 7.9518,Y 109.876,Z 109,A 80.9307,B 24.9302,C -1.9298,E1 25.0128,E2 364.8214} C_DIS
LIN {X 10.798,Y 109.6338,Z 109,A 79.4531,B 24.9302,C -1.93,E1 25.0169,E2 366.2978} C_DIS
LIN {X 13.4853,Y 109.3357,Z 109,A 78.0471,B 24.9302,C -1.9297,E1 25.0208,E2 367.7033} C_DIS
LIN {X 16.0133,Y 108.9934,Z 109,A 76.7433,B 24.9302,C -1.9303,E1 25.0244,E2 369.0045} C_DIS
LIN {X 18.8339,Y 108.5424,Z 109,A 75.2365,B 24.9302,C -1.9289,E1 25.0285,E2 370.513} C_DIS
LIN {X 21.492,Y 108.0475,Z 109,A 73.8315,B 24.9302,C -1.9284,E1 25.0324,E2 371.9177} C_DIS
LIN {X 23.8513,Y 107.5498,Z 109,A 72.5655,B 24.9304,C -1.9273,E1 25.0358,E2 373.1846} C_DIS
LIN {X 26.6194,Y 106.8989,Z 109,A 71.0941,B 24.9304,C -1.9268,E1 25.0398,E2 374.6552} C_DIS
LIN {X 29.3822,Y 106.1737,Z 109,A 69.618,B 24.9304,C -1.9262,E1 25.0438,E2 376.1303} C_DIS
LIN {X 31.8326,Y 105.464,Z 109,A 68.2933,B 24.9305,C -1.9253,E1 25.0473,E2 377.4548} C_DIS
LIN {X 34.4112,Y 104.6511,Z 109,A 66.8893,B 24.9305,C -1.9243,E1 25.0511,E2 378.8586} C_DIS
LIN {X 36.9691,Y 103.775,Z 109,A 65.4857,B 24.9307,C -1.9232,E1 25.0548,E2 380.2621} C_DIS
LIN {X 39.4806,Y 102.8457,Z 109,A 64.086,B 24.9307,C -1.9215,E1 25.0584,E2 381.6626} C_DIS
LIN {X 41.8771,Y 101.8929,Z 109,A 62.7431,B 24.9309,C -1.9201,E1 25.0619,E2 383.0058} C_DIS
LIN {X 44.6431,Y 100.7132,Z 109,A 61.1973,B 24.9309,C -1.9191,E1 25.0659,E2 384.5503} C_DIS
LIN {X 46.9628,Y 99.6517,Z 109,A 59.8739,B 24.9311,C -1.9177,E1 25.0692,E2 385.8737} C_DIS
LIN {X 49.3435,Y 98.4944,Z 109,A 58.4875,B 24.9312,C -1.9156,E1 25.0727,E2 387.2614} C_DIS
LIN {X 51.9311,Y 97.1562,Z 109,A 56.9901,B 24.9313,C -1.9143,E1 25.0764,E2 388.7576} C_DIS
LIN {X 54.2998,Y 95.8525,Z 109,A 55.5881,B 24.9314,C -1.9125,E1 25.0798,E2 390.1598} C_DIS
LIN {X 56.5043,Y 94.5687,Z 109,A 54.2769,B 24.9315,C -1.9112,E1 25.083,E2 391.47} C_DIS
LIN {X 58.8081,Y 93.1535,Z 109,A 52.8897,B 24.9316,C -1.9098,E1 25.0863,E2 392.856} C_DIS
LIN {X 61.0765,Y 91.6823,Z 109,A 51.4623,B 24.9318,C -1.9067,E1 25.0896,E2 394.2861} C_DIS
LIN {X 63.3081,Y 90.1558,Z 109,A 50.054,B 24.932,C -1.9042,E1 25.0928,E2 395.6955} C_DIS
LIN {X 65.6248,Y 88.4847,Z 109,A 48.5812,B 24.9322,C -1.9021,E1 25.0961,E2 397.1679} C_DIS
LIN {X 67.7765,Y 86.8476,Z 109,A 47.1803,B 24.9323,C -1.8998,E1 25.0992,E2 398.5691} C_DIS
LIN {X 69.8875,Y 85.1581,Z 109,A 45.7801,B 24.9325,C -1.8974,E1 25.1023,E2 399.9697} C_DIS
LIN {X 71.9563,Y 83.4173,Z 109,A 44.3795,B 24.9327,C -1.8949,E1 25.1053,E2 401.3707} C_DIS
LIN {X 73.9818,Y 81.6263,Z 109,A 42.9793,B 24.9329,C -1.8924,E1 25.1082,E2 402.7715} C_DIS
LIN {X 75.9627,Y 79.7861,Z 109,A 41.5796,B 24.9331,C -1.8897,E1 25.111,E2 404.1717} C_DIS
LIN {X 77.8979,Y 77.8979,Z 109,A 40.1796,B 24.9332,C -1.887,E1 25.1138,E2 405.5722} C_DIS
LIN {X 79.7861,Y 75.9627,Z 109,A 38.78,B 24.9334,C -1.8842,E1 25.1165,E2 406.9724} C_DIS
LIN {X 81.6263,Y 73.9818,Z 109,A 37.3807,B 24.9336,C -1.8813,E1 25.1192,E2 408.3723} C_DIS
LIN {X 83.1371,Y 72.2772,Z 109,A 36.1535,B 24.934,C -1.8768,E1 25.1214,E2 409.6046} C_DIS
LIN {X 85.1581,Y 69.8874,Z 109,A 34.5823,B 24.934,C -1.8754,E1 25.1242,E2 411.172} C_DIS
LIN {X 86.8476,Y 67.7765,Z 109,A 33.1833,B 24.9343,C -1.8723,E1 25.1267,E2 412.5717} C_DIS
LIN {X 88.3868,Y 65.7552,Z 109,A 31.8607,B 24.9345,C -1.869,E1 25.1289,E2 413.8958} C_DIS
LIN {X 90.0686,Y 63.4335,Z 109,A 30.3857,B 24.9347,C -1.8659,E1 25.1313,E2 415.3708} C_DIS
LIN {X 91.5126,Y 61.3304,Z 109,A 29.059,B 24.935,C -1.8626,E1 25.1334,E2 416.699} C_DIS
LIN {X 93.0726,Y 58.9376,Z 109,A 27.589,B 24.9352,C -1.8593,E1 25.1356,E2 418.1692} C_DIS
LIN {X 94.491,Y 56.6357,Z 109,A 26.1908,B 24.9354,C -1.8559,E1 25.1376,E2 419.5683} C_DIS
LIN {X 95.8525,Y 54.2998,Z 109,A 24.7927,B 24.9357,C -1.8525,E1 25.1396,E2 420.9672} C_DIS
LIN {X 97.0241,Y 52.1745,Z 109,A 23.5158,B 24.936,C -1.8484,E1 25.1413,E2 422.2472} C_DIS
LIN {X 98.3319,Y 49.6671,Z 109,A 22.0687,B 24.9362,C -1.8453,E1 25.1431,E2 423.6938} C_DIS
LIN {X 99.5873,Y 47.1013,Z 109,A 20.5994,B 24.9364,C -1.8418,E1 25.1449,E2 425.1635} C_DIS
LIN {X 100.7132,Y 44.6431,Z 109,A 19.2018,B 24.9367,C -1.8382,E1 25.1465,E2 426.5621} C_DIS
LIN {X 101.7785,Y 42.158,Z 109,A 17.8045,B 24.9369,C -1.8345,E1 25.148,E2 427.9605} C_DIS
LIN {X 102.7266,Y 39.7897,Z 109,A 16.4785,B 24.9372,C -1.8306,E1 25.1494,E2 429.2882} C_DIS
LIN {X 103.7245,Y 37.1132,Z 109,A 15.0093,B 24.9374,C -1.8269,E1 25.1508,E2 430.7579} C_DIS
LIN {X 104.9732,Y 33.4155,Z 109,A 12.9928,B 24.9378,C -1.8214,E1 25.1526,E2 432.776} C_DIS
LIN {X 105.8051,Y 30.6829,Z 109,A 11.5168,B 24.9381,C -1.8173,E1 25.1537,E2 434.2533} C_DIS
LIN {X 106.4864,Y 28.2245,Z 109,A 10.1988,B 24.9383,C -1.8136,E1 25.1547,E2 435.5724} C_DIS
LIN {X 107.1389,Y 25.6358,Z 109,A 8.8613,B 24.9385,C -1.8116,E1 25.1556,E2 436.9069} C_DIS
LIN {X 107.6591,Y 23.3502,Z 109,A 7.5343,B 24.9391,C -1.803,E1 25.1564,E2 438.2464} C_DIS
LIN {X 108.2742,Y 20.3144,Z 109,A 6.0011,B 24.9391,C -1.8014,E1 25.1572,E2 439.7745} C_DIS
LIN {X 108.7401,Y 17.6511,Z 109,A 4.6042,B 24.9394,C -1.7974,E1 25.1579,E2 441.1727} C_DIS
LIN {X 109.1405,Y 14.9772,Z 109,A 3.2076,B 24.9397,C -1.7933,E1 25.1584,E2 442.5706} C_DIS
LIN {X 109.4752,Y 12.2942,Z 109,A 1.818,B 24.94,C -1.7896,E1 25.1589,E2 443.9609} C_DIS
LIN {X 109.744,Y 9.6038,Z 109,A 0.4142,B 24.9403,C -1.7852,E1 25.1593,E2 445.3667} C_DIS
LIN {X 109.9569,Y 6.7553,Z 109,A -1.0536,B 24.9405,C -1.7812,E1 25.1595,E2 446.8353} C_DIS
LIN {X 110.083,Y 4.2074,Z 109,A -2.3789,B 24.9408,C -1.777,E1 25.1597,E2 448.1626} C_DIS
LIN {X 110.1531,Y 1.5046,Z 109,A -3.7808,B 24.9411,C -1.7726,E1 25.1597,E2 449.5664} C_DIS
LIN {X 110.1531,Y -1.5046,Z 109,A -5.2505,B 24.9411,C -1.7718,E1 25.1597,E2 451.0293} C_DIS
LIN {X 110.0943,Y -3.9022,Z 109,A -6.5682,B 24.9416,C -1.7646,E1 25.1597,E2 452.3561} C_DIS
LIN {X 109.9576,Y -6.7435,Z 109,A -8.0293,B 24.9419,C -1.7606,E1 25.1594,E2 453.818} C_DIS
LIN {X 109.7598,Y -9.4298,Z 109,A -9.4212,B 24.9422,C -1.7564,E1 25.1591,E2 455.2115} C_DIS
LIN {X 109.5089,Y -11.9907,Z 109,A -10.7575,B 24.9425,C -1.7522,E1 25.1587,E2 456.5498} C_DIS
LIN {X 109.162,Y -14.826,Z 109,A -12.2253,B 24.9427,C -1.7482,E1 25.1582,E2 458.0184} C_DIS
LIN {X 108.7886,Y -17.3496,Z 109,A -13.5504,B 24.943,C -1.7439,E1 25.1576,E2 459.3457} C_DIS
LIN {X 108.3301,Y -20.0142,Z 109,A -14.9468,B 24.9433,C -1.7398,E1 25.157,E2 460.7436} C_DIS
LIN {X 107.8063,Y -22.6667,Z 109,A -16.3071,B 24.9434,C -1.7374,E1 25.1562,E2 462.1018} C_DIS
LIN {X 107.1832,Y -25.4543,Z 109,A -17.8112,B 24.9438,C -1.7317,E1 25.1553,E2 463.6104} C_DIS
LIN {X 106.5262,Y -28.0771,Z 109,A -19.2081,B 24.9441,C -1.7277,E1 25.1543,E2 465.0089} C_DIS
LIN {X 105.8051,Y -30.6829,Z 109,A -20.6046,B 24.9443,C -1.7236,E1 25.1532,E2 466.407} C_DIS
LIN {X 105.0655,Y -33.1244,Z 109,A -21.9298,B 24.9446,C -1.7195,E1 25.1521,E2 467.7342} C_DIS
LIN {X 104.2209,Y -35.6929,Z 109,A -23.3191,B 24.9448,C -1.7158,E1 25.1509,E2 469.1244} C_DIS
LIN {X 103.3136,Y -38.2398,Z 109,A -24.7236,B 24.9451,C -1.7115,E1 25.1496,E2 470.5312} C_DIS
LIN {X 102.344,Y -40.7637,Z 109,A -26.1204,B 24.9454,C -1.7076,E1 25.1481,E2 471.9296} C_DIS
LIN {X 101.3128,Y -43.2631,Z 109,A -27.5101,B 24.9456,C -1.704,E1 25.1466,E2 473.3201} C_DIS
LIN {X 100.2205,Y -45.7364,Z 109,A -28.9144,B 24.9459,C -1.6998,E1 25.145,E2 474.7267} C_DIS
LIN {X 99.1515,Y -48.0082,Z 109,A -30.2248,B 24.9461,C -1.6957,E1 25.1435,E2 476.0398} C_DIS
LIN {X 97.8556,Y -50.5989,Z 109,A -31.7014,B 24.9463,C -1.6925,E1 25.1416,E2 477.5161} C_DIS
LIN {X 96.5844,Y -52.9852,Z 109,A -33.1062,B 24.9466,C -1.6884,E1 25.1397,E2 478.9231} C_DIS
LIN {X 95.288,Y -55.282,Z 109,A -34.4761,B 24.9468,C -1.6844,E1 25.1378,E2 480.2952} C_DIS
LIN {X 93.8682,Y -57.6605,Z 109,A -35.901,B 24.947,C -1.681,E1 25.1358,E2 481.721} C_DIS
LIN {X 92.4249,Y -59.9468,Z 109,A -37.2913,B 24.9473,C -1.6777,E1 25.1337,E2 483.1122} C_DIS
LIN {X 90.9259,Y -62.197,Z 109,A -38.6889,B 24.9475,C -1.6741,E1 25.1315,E2 484.5113} C_DIS
LIN {X 89.2834,Y -64.534,Z 109,A -40.1657,B 24.9477,C -1.6703,E1 25.1291,E2 485.9897} C_DIS
LIN {X 87.6728,Y -66.7057,Z 109,A -41.5639,B 24.9479,C -1.6669,E1 25.1267,E2 487.3894} C_DIS
LIN {X 86.104,Y -68.7174,Z 109,A -42.883,B 24.9481,C -1.6636,E1 25.1244,E2 488.7099} C_DIS
LIN {X 84.3917,Y -70.8098,Z 109,A -44.2887,B 24.9484,C -1.6599,E1 25.1219,E2 490.1179} C_DIS
LIN {X 82.528,Y -72.9745,Z 109,A -45.7585,B 24.9486,C -1.6568,E1 25.1192,E2 491.5886} C_DIS
LIN {X 80.8155,Y -74.8654,Z 109,A -47.0857,B 24.9488,C -1.6534,E1 25.1167,E2 492.9179} C_DIS
LIN {X 78.8479,Y -76.9361,Z 109,A -48.5563,B 24.949,C -1.6503,E1 25.1139,E2 494.3894} C_DIS
LIN {X 77.0447,Y -78.7406,Z 109,A -49.8761,B 24.9491,C -1.6474,E1 25.1113,E2 495.7105} C_DIS
LIN {X 75.256,Y -80.4507,Z 109,A -51.196,B 24.9494,C -1.6429,E1 25.1086,E2 497.0356} C_DIS
LIN {X 72.9745,Y -82.528,Z 109,A -52.753,B 24.9495,C -1.6412,E1 25.1053,E2 498.5904} C_DIS
LIN {X 71.0435,Y -84.195,Z 109,A -54.0808,B 24.9497,C -1.6382,E1 25.1025,E2 499.9202} C_DIS
LIN {X 68.8372,Y -86.0093,Z 109,A -55.552,B 24.9499,C -1.6355,E1 25.0993,E2 501.3922} C_DIS
LIN {X 66.8266,Y -87.5796,Z 109,A -56.8726,B 24.95,C -1.6329,E1 25.0964,E2 502.714} C_DIS
LIN {X 64.6572,Y -89.1932,Z 109,A -58.2715,B 24.9502,C -1.6302,E1 25.0933,E2 504.1142} C_DIS
LIN {X 62.3234,Y -90.8402,Z 109,A -59.7517,B 24.9504,C -1.6274,E1 25.0899,E2 505.5959} C_DIS
LIN {X 60.0753,Y -92.3424,Z 109,A -61.1519,B 24.9505,C -1.6249,E1 25.0866,E2 506.9975} C_DIS
LIN {X 57.9205,Y -93.708,Z 109,A -62.4784,B 24.9507,C -1.6224,E1 25.0835,E2 508.3257} C_DIS
LIN {X 55.6034,Y -95.1012,Z 109,A -63.8739,B 24.9508,C -1.6203,E1 25.0801,E2 509.7219} C_DIS
LIN {X 53.2527,Y -96.4371,Z 109,A -65.2822,B 24.951,C -1.6176,E1 25.0767,E2 511.1322} C_DIS
LIN {X 50.7349,Y -97.7861,Z 109,A -66.7548,B 24.951,C -1.6156,E1 25.073,E2 512.6054} C_DIS
LIN {X 48.3198,Y -99.0018,Z 109,A -68.1563,B 24.9512,C -1.6135,E1 25.0695,E2 514.0082} C_DIS
LIN {X 46.0141,Y -100.0934,Z 109,A -69.4859,B 24.9514,C -1.6113,E1 25.0661,E2 515.3395} C_DIS
LIN {X 43.7363,Y -101.1085,Z 109,A -70.8077,B 24.9515,C -1.6083,E1 25.0628,E2 516.6653} C_DIS
LIN {X 41.0473,Y -102.2306,Z 109,A -72.2897,B 24.9515,C -1.6075,E1 25.0589,E2 518.1458} C_DIS
LIN {X 38.5261,Y -103.2072,Z 109,A -73.6914,B 24.9517,C -1.6058,E1 25.0553,E2 519.5485} C_DIS
LIN {X 35.8376,Y -104.1721,Z 109,A -75.1655,B 24.9517,C -1.6044,E1 25.0514,E2 521.023} C_DIS
LIN {X 33.4155,Y -104.9732,Z 109,A -76.4963,B 24.9519,C -1.6026,E1 25.0478,E2 522.3556} C_DIS
LIN {X 30.9789,Y -105.7173,Z 109,A -77.826,B 24.9519,C -1.6009,E1 25.0443,E2 523.6869} C_DIS
LIN {X 28.2245,Y -106.4864,Z 109,A -79.2948,B 24.952,C -1.6001,E1 25.0403,E2 525.1553} C_DIS
LIN {X 25.4543,Y -107.1832,Z 109,A -80.777,B 24.9521,C -1.5987,E1 25.0363,E2 526.6386} C_DIS
LIN {X 23.1187,Y -107.7096,Z 109,A -82.0474,B 24.9522,C -1.5965,E1 25.0328,E2 527.9125} C_DIS
LIN {X 20.3144,Y -108.2742,Z 109,A -83.5126,B 24.9522,C -1.5962,E1 25.0288,E2 529.3767} C_DIS
LIN {X 17.6511,Y -108.7401,Z 109,A -84.9164,B 24.9523,C -1.5952,E1 25.025,E2 530.7814} C_DIS
LIN {X 14.9094,Y -109.1502,Z 109,A -86.3467,B 24.9523,C -1.5947,E1 25.021,E2 532.2116} C_DIS
LIN {X 12.2942,Y -109.4752,Z 109,A -87.7252,B 24.9524,C -1.5935,E1 25.0172,E2 533.5919} C_DIS
LIN {X 9.6039,Y -109.744,Z 109,A -89.1114,B 24.9524,C -1.5936,E1 25.0133,E2 534.977} C_DIS
LIN {X 6.7554,Y -109.9569,Z 109,A -90.6064,B 24.9524,C -1.5925,E1 25.0091,E2 536.4739} C_DIS
LIN {X 4.2074,Y -110.083,Z 109,A -91.9398,B 24.9525,C -1.5918,E1 25.0054,E2 537.8087} C_DIS
LIN {X 1.5046,Y -110.1531,Z 109,A -93.3449,B 24.9525,C -1.5914,E1 25.0015,E2 539.2145} C_DIS
LIN {X 1.5046,Y -110.1531,Z 109,A -93.3449,B 24.9525,C -1.5914,E1 25.0015,E2 539.2145} C_DIS
Enddeposition()
LIN {X 0.7629,Y -109.2084,Z 109,A -93.6719,B 24.9514,C -1.6105,E1 25.0007,E2 539.4961} C_DIS
Startdeposition()
$VEL.CP = VEL_PRINT
LIN {X 4.3262,Y -109.126,Z 109,A -91.3271,B 24.9502,C -1.6308,E1 25.0074,E2 537.1036} C_DIS
LIN {X 7.404,Y -108.9599,Z 109,A -89.5173,B 24.9496,C -1.6396,E1 25.0125,E2 535.2737} C_DIS
LIN {X 11.3037,Y -108.6246,Z 109,A -87.4715,B 24.9496,C -1.6404,E1 25.0182,E2 533.2273} C_DIS
LIN {X 15.1474,Y -108.1558,Z 109,A -85.7684,B 24.9503,C -1.6278,E1 25.0228,E2 531.5553} C_DIS
LIN {X 18.1071,Y -107.6997,Z 109,A -83.9046,B 24.9495,C -1.6414,E1 25.028,E2 529.6613} C_DIS
LIN {X 21.7482,Y -107.024,Z 109,A -82.133,B 24.9499,C -1.6357,E1 25.0329,E2 527.9051} C_DIS
LIN {X 24.3942,Y -106.452,Z 109,A -80.7541,B 24.9499,C -1.6353,E1 25.0366,E2 526.5291} C_DIS
LIN {X 27.2164,Y -105.7655,Z 109,A -79.02,B 24.9492,C -1.6458,E1 25.0414,E2 524.7727} C_DIS
LIN {X 30.3609,Y -104.9078,Z 109,A -77.264,B 24.949,C -1.6496,E1 25.0461,E2 523.0106} C_DIS
LIN {X 33.6583,Y -103.8951,Z 109,A -75.5445,B 24.9491,C -1.6479,E1 25.0507,E2 521.2982} C_DIS
LIN {X 37.1134,Y -102.7121,Z 109,A -73.8109,B 24.9494,C -1.6426,E1 25.0552,E2 519.5808} C_DIS
LIN {X 39.1957,Y -101.9366,Z 109,A -72.3431,B 24.9485,C -1.6571,E1 25.0591,E2 518.0817} C_DIS
LIN {X 42.7928,Y -100.479,Z 109,A -70.5293,B 24.949,C -1.6505,E1 25.0637,E2 516.2878} C_DIS
LIN {X 46.3896,Y -98.8695,Z 109,A -68.282,B 24.9483,C -1.6615,E1 25.0695,E2 514.0201} C_DIS
LIN {X 49.9101,Y -97.1396,Z 109,A -66.5787,B 24.949,C -1.6496,E1 25.0737,E2 512.3496} C_DIS
LIN {X 52.82,Y -95.5895,Z 109,A -64.5378,B 24.948,C -1.6661,E1 25.0788,E2 510.2756} C_DIS
LIN {X 55.6321,Y -93.9795,Z 109,A -62.2865,B 24.9463,C -1.6934,E1 25.0843,E2 507.9667} C_DIS
LIN {X 59.2083,Y -91.7688,Z 109,A -60.7383,B 24.9478,C -1.6688,E1 25.0878,E2 506.4816} C_DIS
LIN {X 62.1611,Y -89.7948,Z 109,A -58.774,B 24.9473,C -1.6769,E1 25.0924,E2 504.5047} C_DIS
LIN {X 64.3608,Y -88.2315,Z 109,A -57.2498,B 24.9468,C -1.6847,E1 25.0958,E2 502.9676} C_DIS
LIN {X 67.8323,Y -85.5913,Z 109,A -55.2176,B 24.9472,C -1.6784,E1 25.1003,E2 500.9577} C_DIS
LIN {X 70.3977,Y -83.4959,Z 109,A -53.3058,B 24.9465,C -1.6899,E1 25.1044,E2 499.026} C_DIS
LIN {X 73.1999,Y -81.0498,Z 109,A -51.4176,B 24.9464,C -1.6917,E1 25.1084,E2 497.1412} C_DIS
LIN {X 75.8888,Y -78.5365,Z 109,A -49.5531,B 24.9463,C -1.6934,E1 25.1121,E2 495.2803} C_DIS
LIN {X 78.5342,Y -75.8912,Z 109,A -47.8405,B 24.9467,C -1.6872,E1 25.1154,E2 493.5896} C_DIS
LIN {X 80.5207,Y -73.7801,Z 109,A -46.1051,B 24.9458,C -1.7005,E1 25.1188,E2 491.8304} C_DIS
LIN {X 82.2048,Y -71.8989,Z 109,A -44.6787,B 24.9453,C -1.7084,E1 25.1214,E2 490.3917} C_DIS
LIN {X 85.7286,Y -67.6587,Z 109,A -41.9535,B 24.9453,C -1.7087,E1 25.1262,E2 487.6785} C_DIS
LIN {X 87.7249,Y -65.0525,Z 109,A -40.1591,B 24.9448,C -1.7165,E1 25.1293,E2 485.8742} C_DIS
LIN {X 89.6185,Y -62.4148,Z 109,A -38.4922,B 24.9446,C -1.7197,E1 25.132,E2 484.2079} C_DIS
LIN {X 92.8971,Y -57.4236,Z 109,A -35.2201,B 24.9436,C -1.7348,E1 25.1369,E2 480.9167} C_DIS
LIN {X 95.0431,Y -53.7986,Z 109,A -32.6368,B 24.9421,C -1.758,E1 25.1406,E2 478.292} C_DIS
LIN {X 96.9311,Y -50.3175,Z 109,A -31.0265,B 24.9431,C -1.7432,E1 25.1426,E2 476.7251} C_DIS
LIN {X 99.217,Y -45.6431,Z 109,A -28.2777,B 24.9425,C -1.7523,E1 25.1459,E2 473.9697} C_DIS
LIN {X 100.4573,Y -42.8443,Z 109,A -26.7143,B 24.9423,C -1.7553,E1 25.1476,E2 472.4077} C_DIS
LIN {X 101.9388,Y -39.19,Z 109,A -24.6555,B 24.9419,C -1.7612,E1 25.1497,E2 470.3463} C_DIS
LIN {X 103.4144,Y -35.1081,Z 109,A -22.4559,B 24.9416,C -1.7649,E1 25.1518,E2 468.1504} C_DIS
LIN {X 104.3015,Y -32.3771,Z 109,A -20.6533,B 24.9404,C -1.783,E1 25.1533,E2 466.3154} C_DIS
LIN {X 105.6542,Y -27.6494,Z 109,A -18.3888,B 24.9408,C -1.777,E1 25.155,E2 464.078} C_DIS
LIN {X 106.449,Y -24.4074,Z 109,A -16.724,B 24.9407,C -1.7787,E1 25.156,E2 462.4187} C_DIS
LIN {X 107.1315,Y -21.2193,Z 109,A -14.8134,B 24.9397,C -1.7932,E1 25.1571,E2 460.4852} C_DIS
LIN {X 107.8668,Y -17.0881,Z 109,A -12.7714,B 24.9397,C -1.7932,E1 25.158,E2 458.4552} C_DIS
LIN {X 108.3807,Y -13.4549,Z 109,A -10.771,B 24.9391,C -1.8028,E1 25.1588,E2 456.444} C_DIS
LIN {X 108.785,Y -9.6466,Z 109,A -8.8437,B 24.9389,C -1.8057,E1 25.1593,E2 454.5214} C_DIS
LIN {X 108.9939,Y -6.9008,Z 109,A -7.5041,B 24.9389,C -1.8057,E1 25.1595,E2 453.1898} C_DIS
LIN {X 109.1424,Y -3.8978,Z 109,A -5.8893,B 24.9384,C -1.8124,E1 25.1597,E2 451.5685} C_DIS
LIN {X 109.2109,Y -0.4008,Z 109,A -4.103,B 24.9382,C -1.8162,E1 25.1597,E2 449.7839} C_DIS
LIN {X 109.1557,Y 3.4806,Z 109,A -2.2356,B 24.9382,C -1.8152,E1 25.1597,E2 447.9299} C_DIS
LIN {X 109.001,Y 6.7957,Z 109,A -0.1972,B 24.9369,C -1.8341,E1 25.1594,E2 445.8591} C_DIS
LIN {X 108.7017,Y 10.549,Z 109,A 1.6273,B 24.9369,C -1.8337,E1 25.1589,E2 444.0463} C_DIS
LIN {X 108.286,Y 14.1862,Z 109,A 3.4071,B 24.9369,C -1.8336,E1 25.1583,E2 442.2774} C_DIS
LIN {X 107.9235,Y 16.7213,Z 109,A 4.8918,B 24.9363,C -1.8442,E1 25.1577,E2 440.7765} C_DIS
LIN {X 107.4673,Y 19.4389,Z 109,A 6.7219,B 24.9347,C -1.8659,E1 25.1568,E2 438.9057} C_DIS
LIN {X 106.8018,Y 22.8181,Z 109,A 8.1572,B 24.9355,C -1.8549,E1 25.156,E2 437.5048} C_DIS
LIN {X 106.1084,Y 25.8471,Z 109,A 9.7371,B 24.9353,C -1.8577,E1 25.155,E2 435.9274} C_DIS
LIN {X 104.507,Y 31.7141,Z 109,A 13.0195,B 24.9343,C -1.8715,E1 25.1525,E2 432.6313} C_DIS
LIN {X 103.4369,Y 35.0415,Z 109,A 14.6979,B 24.9344,C -1.8702,E1 25.151,E2 430.9656} C_DIS
LIN {X 102.1666,Y 38.5885,Z 109,A 16.5998,B 24.9343,C -1.8727,E1 25.1492,E2 429.0683} C_DIS
LIN {X 100.9458,Y 41.6812,Z 109,A 18.326,B 24.934,C -1.877,E1 25.1474,E2 427.3414} C_DIS
LIN {X 99.9059,Y 44.1152,Z 109,A 20.9171,B 24.9298,C -1.9347,E1 25.1443,E2 424.6284} C_DIS
LIN {X 97.1747,Y 49.8414,Z 109,A 23.0725,B 24.9329,C -1.8917,E1 25.1417,E2 422.586} C_DIS
LIN {X 95.3691,Y 53.2147,Z 109,A 25.035,B 24.9327,C -1.8952,E1 25.1391,E2 420.6254} C_DIS
LIN {X 93.6758,Y 56.1459,Z 109,A 26.8584,B 24.9322,C -1.902,E1 25.1365,E2 418.7953} C_DIS
LIN {X 92.3366,Y 58.3208,Z 109,A 28.3282,B 24.9315,C -1.9113,E1 25.1343,E2 417.3111} C_DIS
LIN {X 90.6294,Y 60.9387,Z 109,A 29.8785,B 24.9315,C -1.9116,E1 25.1319,E2 415.7678} C_DIS
LIN {X 88.5567,Y 63.9146,Z 109,A 31.6589,B 24.9315,C -1.911,E1 25.1291,E2 413.9974} C_DIS
LIN {X 86.5798,Y 66.5659,Z 109,A 33.1964,B 24.9318,C -1.9067,E1 25.1265,E2 412.4774} C_DIS
LIN {X 84.7415,Y 68.8911,Z 109,A 35.0566,B 24.9306,C -1.9238,E1 25.1232,E2 410.5857} C_DIS
LIN {X 82.4588,Y 71.6081,Z 109,A 36.8907,B 24.9304,C -1.9269,E1 25.1199,E2 408.7526} C_DIS
LIN {X 80.3287,Y 73.9893,Z 109,A 38.6314,B 24.9299,C -1.9335,E1 25.1166,E2 407.0039} C_DIS
LIN {X 77.8079,Y 76.6357,Z 109,A 40.4122,B 24.93,C -1.9317,E1 25.1131,E2 405.2349} C_DIS
LIN {X 75.4938,Y 78.9172,Z 109,A 42.2421,B 24.9294,C -1.9407,E1 25.1094,E2 403.3913} C_DIS
LIN {X 72.7442,Y 81.4578,Z 109,A 43.9701,B 24.9298,C -1.9345,E1 25.1059,E2 401.685} C_DIS
LIN {X 70.3188,Y 83.563,Z 109,A 45.9165,B 24.9288,C -1.9491,E1 25.1017,E2 399.7119} C_DIS
LIN {X 67.0749,Y 86.1876,Z 109,A 47.8001,B 24.9294,C -1.94,E1 25.0977,E2 397.8568} C_DIS
LIN {X 64.8115,Y 87.9015,Z 109,A 49.4176,B 24.9288,C -1.9481,E1 25.094,E2 396.2258} C_DIS
LIN {X 62.0892,Y 89.8449,Z 109,A 51.2511,B 24.9284,C -1.9545,E1 25.0898,E2 394.3835} C_DIS
LIN {X 59.402,Y 91.6445,Z 109,A 52.9573,B 24.9282,C -1.9576,E1 25.0858,E2 392.6756} C_DIS
LIN {X 55.9936,Y 93.7658,Z 109,A 56.0877,B 24.9246,C -2.0049,E1 25.0781,E2 389.4431} C_DIS
LIN {X 50.3921,Y 96.8918,Z 109,A 58.3692,B 24.9278,C -1.9628,E1 25.0727,E2 387.2676} C_DIS
LIN {X 46.8593,Y 98.6485,Z 109,A 60.4297,B 24.9276,C -1.965,E1 25.0675,E2 385.2074} C_DIS
LIN {X 44.2149,Y 99.8624,Z 109,A 62.0583,B 24.9272,C -1.971,E1 25.0634,E2 383.5685} C_DIS
LIN {X 40.3761,Y 101.4745,Z 109,A 63.9413,B 24.9279,C -1.9606,E1 25.0586,E2 381.7145} C_DIS
LIN {X 37.2833,Y 102.6501,Z 109,A 65.874,B 24.9272,C -1.9705,E1 25.0535,E2 379.7624} C_DIS
LIN {X 33.946,Y 103.802,Z 109,A 67.6791,B 24.9272,C -1.9701,E1 25.0487,E2 377.9618} C_DIS
LIN {X 27.9938,Y 105.5636,Z 109,A 70.8421,B 24.9274,C -1.9685,E1 25.0402,E2 374.808} C_DIS
LIN {X 24.8409,Y 106.3488,Z 109,A 72.5612,B 24.9272,C -1.97,E1 25.0356,E2 373.0877} C_DIS
LIN {X 22.3631,Y 106.8978,Z 109,A 74.1484,B 24.9264,C -1.9813,E1 25.0312,E2 371.4759} C_DIS
LIN {X 18.021,Y 107.714,Z 109,A 76.2602,B 24.927,C -1.9736,E1 25.0254,E2 369.3845} C_DIS
LIN {X 14.6664,Y 108.2237,Z 109,A 78.1731,B 24.9265,C -1.9795,E1 25.0201,E2 367.4593} C_DIS
LIN {X 10.7096,Y 108.6868,Z 109,A 80.2465,B 24.9265,C -1.9792,E1 25.0143,E2 365.3881} C_DIS
LIN {X 7.377,Y 108.9617,Z 109,A 81.8451,B 24.927,C -1.9729,E1 25.0099,E2 363.8052} C_DIS
LIN {X 3.8522,Y 109.1443,Z 109,A 83.5814,B 24.9274,C -1.9681,E1 25.0051,E2 362.0809} C_DIS
LIN {X 0.6096,Y 109.2095,Z 109,A 85.4959,B 24.9268,C -1.9765,E1 24.9997,E2 360.1466} C_DIS
LIN {X -2.3491,Y 109.1864,Z 109,A 86.9338,B 24.9271,C -1.9715,E1 24.9957,E2 358.7206} C_DIS
LIN {X -6.4692,Y 109.0203,Z 109,A 89.1131,B 24.9271,C -1.9713,E1 24.9897,E2 356.5411} C_DIS
LIN {X -9.8179,Y 108.7692,Z 109,A 90.9296,B 24.9271,C -1.9727,E1 24.9846,E2 354.7204} C_DIS
LIN {X -13.1896,Y 108.4129,Z 109,A 92.5346,B 24.9276,C -1.9647,E1 24.9802,E2 353.1334} C_DIS
LIN {X -16.6605,Y 107.9329,Z 109,A 94.5113,B 24.9273,C -1.9691,E1 24.9747,E2 351.1447} C_DIS
LIN {X -23.659,Y 106.6184,Z 109,A 98.3812,B 24.9271,C -1.9714,E1 24.9641,E2 347.2651} C_DIS
LIN {X -26.1938,Y 106.0239,Z 109,A 100.2286,B 24.9258,C -1.9894,E1 24.9589,E2 345.3723} C_DIS
LIN {X -30.114,Y 104.9778,Z 109,A 101.8646,B 24.9274,C -1.9673,E1 24.9547,E2 343.7861} C_DIS
LIN {X -33.6572,Y 103.8955,Z 109,A 103.7575,B 24.9277,C -1.9631,E1 24.9496,E2 341.8999} C_DIS
LIN {X -39.9012,Y 101.6611,Z 109,A 107.212,B 24.9282,C -1.9575,E1 24.9406,E2 338.4516} C_DIS
LIN {X -43.2966,Y 100.2628,Z 109,A 109.2226,B 24.9282,C -1.9581,E1 24.9354,E2 336.4351} C_DIS
LIN {X -46.7851,Y 98.6841,Z 109,A 111.0508,B 24.9289,C -1.9479,E1 24.9308,E2 334.6266} C_DIS
LIN {X -50.0255,Y 97.0807,Z 109,A 113.0211,B 24.9289,C -1.9477,E1 24.9259,E2 332.6515} C_DIS
LIN {X -53.1089,Y 95.4282,Z 109,A 114.7613,B 24.9294,C -1.9408,E1 24.9217,E2 330.9227} C_DIS
LIN {X -55.8784,Y 93.834,Z 109,A 116.7439,B 24.9287,C -1.9497,E1 24.9168,E2 328.913} C_DIS
LIN {X -59.0807,Y 91.8507,Z 109,A 118.5612,B 24.9295,C -1.9398,E1 24.9126,E2 327.1134} C_DIS
LIN {X -61.8957,Y 89.9793,Z 109,A 120.5677,B 24.929,C -1.9453,E1 24.9079,E2 325.0871} C_DIS
LIN {X -65.3983,Y 87.4654,Z 109,A 122.6279,B 24.93,C -1.9329,E1 24.9033,E2 323.0494} C_DIS
LIN {X -70.0429,Y 83.7924,Z 109,A 126.3792,B 24.9286,C -1.9511,E1 24.8951,E2 319.2406} C_DIS
LIN {X -73.2526,Y 81.0022,Z 109,A 127.9555,B 24.9309,C -1.9205,E1 24.8919,E2 317.7307} C_DIS
LIN {X -78.1998,Y 76.2381,Z 109,A 132.3773,B 24.9292,C -1.9434,E1 24.883,E2 313.2357} C_DIS
LIN {X -81.3993,Y 72.8095,Z 109,A 134.0949,B 24.9317,C -1.9086,E1 24.8799,E2 311.5936} C_DIS
LIN {X -83.5532,Y 70.3299,Z 109,A 135.9652,B 24.9317,C -1.9097,E1 24.8765,E2 309.712} C_DIS
LIN {X -86.0774,Y 67.2173,Z 109,A 138.0789,B 24.932,C -1.9045,E1 24.8728,E2 307.6007} C_DIS
LIN {X -87.8212,Y 64.9212,Z 109,A 139.5139,B 24.9325,C -1.8975,E1 24.8705,E2 306.1756} C_DIS
LIN {X -90.056,Y 61.7854,Z 109,A 141.8356,B 24.9321,C -1.9034,E1 24.8667,E2 303.8284} C_DIS
LIN {X -92.5158,Y 58.034,Z 109,A 143.6435,B 24.934,C -1.876,E1 24.8641,E2 302.0766} C_DIS
LIN {X -94.2348,Y 55.2002,Z 109,A 145.7452,B 24.9334,C -1.8847,E1 24.861,E2 299.9433} C_DIS
LIN {X -95.7797,Y 52.4741,Z 109,A 147.3722,B 24.9338,C -1.8793,E1 24.8588,E2 298.3207} C_DIS
LIN {X -97.1881,Y 49.8153,Z 109,A 148.847,B 24.9344,C -1.8707,E1 24.8569,E2 296.8586} C_DIS
LIN {X -99.9479,Y 44.018,Z 109,A 152.3976,B 24.9346,C -1.8674,E1 24.8528,E2 293.2965} C_DIS
LIN {X -101.5255,Y 40.2463,Z 109,A 154.2475,B 24.9359,C -1.8496,E1 24.8508,E2 291.4786} C_DIS
LIN {X -102.3331,Y 38.1487,Z 109,A 155.7712,B 24.9352,C -1.859,E1 24.8493,E2 289.924} C_DIS
LIN {X -103.7522,Y 34.0998,Z 109,A 157.7126,B 24.9365,C -1.8402,E1 24.8476,E2 288.0162} C_DIS
LIN {X -104.4521,Y 31.8914,Z 109,A 159.2179,B 24.936,C -1.8473,E1 24.8463,E2 286.4853} C_DIS
LIN {X -105.3378,Y 28.8296,Z 109,A 160.6623,B 24.937,C -1.8335,E1 24.8453,E2 285.0657} C_DIS
LIN {X -105.9885,Y 26.3388,Z 109,A 162.0463,B 24.9372,C -1.8304,E1 24.8443,E2 283.6808} C_DIS
LIN {X -106.6665,Y 23.4383,Z 109,A 163.6209,B 24.9375,C -1.8259,E1 24.8433,E2 282.1079} C_DIS
LIN {X -107.1851,Y 20.9407,Z 109,A 164.877,B 24.938,C -1.8185,E1 24.8426,E2 280.8619} C_DIS
LIN {X -107.6098,Y 18.6444,Z 109,A 166.202,B 24.938,C -1.8183,E1 24.842,E2 279.5296} C_DIS
LIN {X -108.4274,Y 13.0653,Z 109,A 169.2939,B 24.9383,C -1.8137,E1 24.8408,E2 276.4301} C_DIS
LIN {X -108.7359,Y 10.1779,Z 109,A 171.5221,B 24.9368,C -1.8356,E1 24.8402,E2 274.1364} C_DIS
LIN {X -109.0739,Y 5.4982,Z 109,A 173.2127,B 24.9394,C -1.7983,E1 24.84,E2 272.5246} C_DIS
LIN {X -109.1893,Y 2.1938,Z 109,A 175.0501,B 24.9395,C -1.7965,E1 24.8398,E2 270.6803} C_DIS
LIN {X -109.2113,Y -0.3309,Z 109,A 176.7269,B 24.9389,C -1.8056,E1 24.8398,E2 268.9718} C_DIS
LIN {X -109.0398,Y -6.1158,Z 109,A 179.3834,B 24.9405,C -1.7814,E1 24.8401,E2 266.357} C_DIS
LIN {X -108.7869,Y -9.6254,Z 109,A -178.6594,B 24.9406,C -1.7797,E1 24.8405,E2 264.3921} C_DIS
LIN {X -108.2215,Y -14.6741,Z 109,A -175.8127,B 24.9407,C -1.7781,E1 24.8415,E2 261.5322} C_DIS
LIN {X -107.3656,Y -20.0036,Z 109,A -173.0488,B 24.9415,C -1.7665,E1 24.8428,E2 258.7795} C_DIS
LIN {X -106.6391,Y -23.5639,Z 109,A -171.1619,B 24.942,C -1.7599,E1 24.8439,E2 256.8973} C_DIS
LIN {X -105.8097,Y -27.0444,Z 109,A -169.6147,B 24.9432,C -1.7415,E1 24.8449,E2 255.3848} C_DIS
LIN {X -105.2087,Y -29.2994,Z 109,A -168.038,B 24.9425,C -1.7512,E1 24.8461,E2 253.776} C_DIS
LIN {X -104.0681,Y -33.1236,Z 109,A -166.1806,B 24.9435,C -1.7358,E1 24.8476,E2 251.9445} C_DIS
LIN {X -102.9386,Y -36.4805,Z 109,A -164.2159,B 24.9436,C -1.7343,E1 24.8494,E2 249.9721} C_DIS
LIN {X -101.7146,Y -39.7649,Z 109,A -162.2949,B 24.9438,C -1.732,E1 24.8513,E2 248.0458} C_DIS
LIN {X -100.4905,Y -42.7655,Z 109,A -160.2672,B 24.9433,C -1.7397,E1 24.8536,E2 245.9886} C_DIS
LIN {X -98.7245,Y -46.7011,Z 109,A -158.3402,B 24.9445,C -1.7203,E1 24.8558,E2 244.0974} C_DIS
LIN {X -97.2691,Y -49.6567,Z 109,A -156.6037,B 24.9448,C -1.7158,E1 24.8579,E2 242.3622} C_DIS
LIN {X -95.5357,Y -52.9164,Z 109,A -154.7098,B 24.9453,C -1.7088,E1 24.8604,E2 240.4749} C_DIS
LIN {X -94.0012,Y -55.5954,Z 109,A -152.6511,B 24.9445,C -1.7214,E1 24.8634,E2 238.3754} C_DIS
LIN {X -92.3069,Y -58.3685,Z 109,A -151.3675,B 24.9458,C -1.7006,E1 24.8653,E2 237.1349} C_DIS
LIN {X -90.5937,Y -60.9913,Z 109,A -149.8992,B 24.9465,C -1.6897,E1 24.8675,E2 235.6853} C_DIS
LIN {X -88.9701,Y -63.3358,Z 109,A -148.085,B 24.946,C -1.6982,E1 24.8704,E2 233.842} C_DIS
LIN {X -86.6278,Y -66.5037,Z 109,A -146.3171,B 24.947,C -1.6815,E1 24.8733,E2 232.1053} C_DIS
LIN {X -84.984,Y -68.5919,Z 109,A -144.8222,B 24.947,C -1.6821,E1 24.876,E2 230.602} C_DIS
LIN {X -83.1436,Y -70.8111,Z 109,A -143.4185,B 24.9475,C -1.6743,E1 24.8784,E2 229.2103} C_DIS
LIN {X -81.2884,Y -72.9335,Z 109,A -141.57,B 24.9468,C -1.6853,E1 24.8819,E2 227.3273} C_DIS
LIN {X -78.1877,Y -76.2507,Z 109,A -139.1337,B 24.947,C -1.6822,E1 24.8866,E2 224.8879} C_DIS
LIN {X -75.2839,Y -79.119,Z 109,A -136.9819,B 24.9472,C -1.6781,E1 24.8909,E2 222.7368} C_DIS
LIN {X -72.4176,Y -81.7502,Z 109,A -134.9234,B 24.9474,C -1.6747,E1 24.8952,E2 220.6781} C_DIS
LIN {X -69.4479,Y -84.2868,Z 109,A -132.8669,B 24.9477,C -1.6711,E1 24.8996,E2 218.6223} C_DIS
LIN {X -66.814,Y -86.3887,Z 109,A -131.3618,B 24.9485,C -1.6575,E1 24.9029,E2 217.1441} C_DIS
LIN {X -64.7887,Y -87.9182,Z 109,A -129.869,B 24.9483,C -1.6616,E1 24.9062,E2 215.6363} C_DIS
LIN {X -62.1188,Y -89.8243,Z 109,A -128.0387,B 24.9482,C -1.6631,E1 24.9105,E2 213.7962} C_DIS
LIN {X -59.1922,Y -91.7792,Z 109,A -125.2899,B 24.9461,C -1.6965,E1 24.9172,E2 210.9591} C_DIS
LIN {X -54.1482,Y -94.8427,Z 109,A -123.0945,B 24.9486,C -1.6556,E1 24.9222,E2 208.8542} C_DIS
LIN {X -50.9918,Y -96.576,Z 109,A -121.3312,B 24.9491,C -1.6481,E1 24.9265,E2 207.104} C_DIS
LIN {X -48.6425,Y -97.7804,Z 109,A -120.0838,B 24.9496,C -1.6408,E1 24.9296,E2 205.8705} C_DIS
LIN {X -45.952,Y -99.0733,Z 109,A -118.4295,B 24.9494,C -1.6425,E1 24.9338,E2 204.208} C_DIS
LIN {X -42.8524,Y -100.4539,Z 109,A -116.4593,B 24.9491,C -1.6482,E1 24.9389,E2 202.2196} C_DIS
LIN {X -39.0594,Y -101.9883,Z 109,A -114.5937,B 24.9499,C -1.6348,E1 24.9436,E2 200.3819} C_DIS
LIN {X -36.284,Y -103.0076,Z 109,A -112.861,B 24.9496,C -1.6408,E1 24.9482,E2 198.6315} C_DIS
LIN {X -30.5952,Y -104.8391,Z 109,A -109.7675,B 24.9498,C -1.6366,E1 24.9565,E2 195.5423} C_DIS
LIN {X -27.2835,Y -105.7483,Z 109,A -107.9031,B 24.9498,C -1.6381,E1 24.9615,E2 193.6716} C_DIS
LIN {X -22.8226,Y -106.8008,Z 109,A -105.4081,B 24.9496,C -1.6406,E1 24.9683,E2 191.1674} C_DIS
LIN {X -19.8171,Y -107.3993,Z 109,A -104.0218,B 24.9502,C -1.6309,E1 24.9721,E2 189.8027} C_DIS
LIN {X -16.6099,Y -107.9407,Z 109,A -102.2905,B 24.9502,C -1.6314,E1 24.9769,E2 188.0685} C_DIS
LIN {X -13.3683,Y -108.3919,Z 109,A -100.3765,B 24.9496,C -1.6392,E1 24.9822,E2 186.1346} C_DIS
LIN {X -10.1459,Y -108.7389,Z 109,A -98.7002,B 24.9497,C -1.6381,E1 24.9869,E2 184.46} C_DIS
LIN {X -6.7851,Y -109.0017,Z 109,A -96.8587,B 24.9495,C -1.6412,E1 24.992,E2 182.6106} C_DIS
LIN {X -3.488,Y -109.1555,Z 109,A -95.2249,B 24.9498,C -1.6373,E1 24.9966,E2 180.9858} C_DIS
LIN {X -0.34,Y -109.2111,Z 109,A -93.7214,B 24.9501,C -1.6314,E1 25.0007,E2 179.4961} C_DIS
LIN {X -0.34,Y -109.2111,Z 109,A -93.7214,B 24.9501,C -1.6314,E1 25.0007,E2 179.4961} C_DIS
Enddeposition()
LIN {X 0.7592,Y -108.2524,Z 109,A -93.6306,B 24.9503,C -1.6281,E1 25.0009,E2 179.4131} C_DIS
Startdeposition()
$VEL.CP = VEL_PRINT
LIN {X -2.3376,Y -108.2354,Z 109,A -95.4658,B 24.9508,C -1.6197,E1 24.9958,E2 181.2684} C_DIS
LIN {X -5.7963,Y -108.105,Z 109,A -97.3393,B 24.951,C -1.6178,E1 24.9905,E2 183.1467} C_DIS
LIN {X -9.4938,Y -107.844,Z 109,A -99.4238,B 24.9513,C -1.6129,E1 24.9847,E2 185.2438} C_DIS
LIN {X -12.5244,Y -107.5332,Z 109,A -100.886,B 24.9509,C -1.6192,E1 24.9807,E2 186.692} C_DIS
LIN {X -15.5653,Y -107.1359,Z 109,A -102.5385,B 24.9509,C -1.6183,E1 24.9761,E2 188.3478} C_DIS
LIN {X -19.62,Y -106.4684,Z 109,A -104.7906,B 24.9511,C -1.6159,E1 24.9699,E2 190.6078} C_DIS
LIN {X -24.861,Y -105.3681,Z 109,A -107.6698,B 24.9511,C -1.6155,E1 24.962,E2 193.4918} C_DIS
Enddeposition()
END
